LIN {X 0,Y 387.005,Z 815.122,A -85,B 0,C 180,E1 -12042.119,E2 -12042.119} C_VEL
LIN {X 0,Y 389.594,Z 822.975,A -85,B 0,C 180,E1 -12042.96,E2 -12042.96} C_VEL
LIN {X 0,Y 390.009,Z 825.761,A -85,B 0,C 180,E1 -12043.242,E2 -12043.242} C_VEL
LIN {X 0,Y 389.304,Z 834.795,A -85,B 0,C 180,E1 -12044.101,E2 -12044.101} C_VEL
LIN {X 0,Y 388.401,Z 845.399,A -85,B 0,C 180,E1 -12045.326,E2 -12045.326} C_VEL
LIN {X 0,Y 387.347,Z 856.042,A -85,B 0,C 180,E1 -12046.891,E2 -12046.891} C_VEL
LIN {X 0,Y 386.493,Z 863.14,A -85,B 0,C 180,E1 -12048.196,E2 -12048.196} C_VEL
LIN {X 0,Y 385.858,Z 869.08,A -85,B 0,C 180,E1 -12049.506,E2 -12049.506} C_VEL
LIN {X 0,Y 385.357,Z 873.167,A -85,B 0,C 180,E1 -12050.553,E2 -12050.553} C_VEL
LIN {X 0,Y 384.731,Z 878.114,A -85,B 0,C 180,E1 -12052.125,E2 -12052.125} C_VEL
LIN {X 0,Y 383.96,Z 881.899,A -85,B 0,C 180,E1 -12053.695,E2 -12053.695} C_VEL
LIN {X 0,Y 383.86,Z 883.852,A -85,B 0,C 180,E1 -12054.748,E2 -12054.748} C_VEL
LIN {X 0,Y 383.471,Z 886.332,A -85,B 0,C 180,E1 -12056.848,E2 -12056.848} C_VEL
LIN {X 0,Y 383.299,Z 887.036,A -85,B 0,C 180,E1 -12057.898,E2 -12057.898} C_VEL
LIN {X 0,Y 383.093,Z 887.297,A -85,B 0,C 180,E1 -12058.949,E2 -12058.949} C_VEL
LIN {X 0,Y 383.035,Z 886.513,A -85,B 0,C 180,E1 -12061.051,E2 -12061.051} C_VEL
LIN {X 0,Y 382.901,Z 884.089,A -85,B 0,C 180,E1 -12063.157,E2 -12063.157} C_VEL
LIN {X 0,Y 383.149,Z 881.129,A -85,B 0,C 180,E1 -12064.735,E2 -12064.735} C_VEL
LIN {X 0,Y 383.443,Z 877.126,A -85,B 0,C 180,E1 -12066.314,E2 -12066.314} C_VEL
LIN {X 0,Y 383.766,Z 871.975,A -85,B 0,C 180,E1 -12067.895,E2 -12067.895} C_VEL
LIN {X 0,Y 384.086,Z 866.854,A -85,B 0,C 180,E1 -12069.187,E2 -12069.187} C_VEL
LIN {X 0,Y 384.606,Z 859.101,A -85,B 0,C 180,E1 -12070.795,E2 -12070.795} C_VEL
LIN {X 0,Y 385.028,Z 851.181,A -85,B 0,C 180,E1 -12072.117,E2 -12072.117} C_VEL
LIN {X 0,Y 385.562,Z 843.782,A -85,B 0,C 180,E1 -12073.171,E2 -12073.171} C_VEL
LIN {X 0,Y 386.012,Z 836.271,A -85,B 0,C 180,E1 -12074.094,E2 -12074.094} C_VEL
LIN {X 0,Y 386.607,Z 826.481,A -85,B 0,C 180,E1 -12075.117,E2 -12075.117} C_VEL
LIN {X 0,Y 386.907,Z 820.016,A -85,B 0,C 180,E1 -12075.69,E2 -12075.69} C_VEL
LIN {X 0,Y 384.066,Z 808.559,A -85,B 0,C 180,E1 -12076.657,E2 -12076.657} C_VEL
LIN {X 0,Y 383.065,Z 804.769,A -85,B 0,C 180,E1 -12076.968,E2 -12076.968} C_VEL
LIN {X 0,Y 383.009,Z 804.767,A -85,B 0,C 180,E1 -12080.636,E2 -12080.636} C_VEL
LIN {X 0,Y 383.012,Z 804.777,A -85,B 0,C 180,E1 -12083.809,E2 -12083.809} C_VEL
LIN {X 0,Y 382.972,Z 804.773,A -85,B 0,C 180,E1 -12087.309,E2 -12087.309} C_VEL
LIN {X 0,Y 382.987,Z 804.773,A -85,B 0,C 180,E1 -12090.918,E2 -12090.918} C_VEL
LIN {X 0,Y 383.018,Z 804.77,A -85,B 0,C 180,E1 -12094.668,E2 -12094.668} C_VEL
LIN {X 0,Y 382.998,Z 804.772,A -85,B 0,C 180,E1 -12097.901,E2 -12097.901} C_VEL
LIN {X 0,Y 382.967,Z 804.777,A -85,B 0,C 180,E1 -12101.35,E2 -12101.35} C_VEL
LIN {X 0,Y 383,Z 804.777,A -85,B 0,C 180,E1 -12104.302,E2 -12104.302} C_VEL
LIN {X 0,Y 383.017,Z 804.77,A -85,B 0,C 180,E1 -12107.239,E2 -12107.239} C_VEL
LIN {X 0,Y 382.992,Z 804.778,A -85,B 0,C 180,E1 -12110.418,E2 -12110.418} C_VEL
LIN {X 0,Y 383.03,Z 804.773,A -85,B 0,C 180,E1 -12114.043,E2 -12114.043} C_VEL
LIN {X 0,Y 382.994,Z 804.774,A -85,B 0,C 180,E1 -12117.577,E2 -12117.577} C_VEL
LIN {X 0,Y 382.999,Z 804.774,A -85,B 0,C 180,E1 -12120.299,E2 -12120.299} C_VEL
LIN {X 0,Y 383.086,Z 804.762,A -85,B 0,C 180,E1 -12124.02,E2 -12124.02} C_VEL
LIN {X 0,Y 383.018,Z 804.772,A -85,B 0,C 180,E1 -12127.334,E2 -12127.334} C_VEL
LIN {X 0,Y 383.066,Z 804.775,A -85,B 0,C 180,E1 -12130.715,E2 -12130.715} C_VEL
LIN {X 0,Y 383.075,Z 804.773,A -85,B 0,C 180,E1 -12131.917,E2 -12131.917} C_VEL
LIN {X 0,Y 386.733,Z 816.026,A -85,B 0,C 180,E1 -12132.822,E2 -12132.822} C_VEL
LIN {X 0,Y 388.874,Z 823.669,A -85,B 0,C 180,E1 -12133.533,E2 -12133.533} C_VEL
LIN {X 0,Y 388.161,Z 834.358,A -85,B 0,C 180,E1 -12134.509,E2 -12134.509} C_VEL
LIN {X 0,Y 387.355,Z 844.687,A -85,B 0,C 180,E1 -12135.686,E2 -12135.686} C_VEL
LIN {X 0,Y 386.66,Z 853.102,A -85,B 0,C 180,E1 -12136.866,E2 -12136.866} C_VEL
LIN {X 0,Y 385.851,Z 860.859,A -85,B 0,C 180,E1 -12138.174,E2 -12138.174} C_VEL
LIN {X 0,Y 385.124,Z 868.416,A -85,B 0,C 180,E1 -12139.75,E2 -12139.75} C_VEL
LIN {X 0,Y 384.606,Z 874.215,A -85,B 0,C 180,E1 -12141.259,E2 -12141.259} C_VEL
LIN {X 0,Y 384.195,Z 878.536,A -85,B 0,C 180,E1 -12142.641,E2 -12142.641} C_VEL
LIN {X 0,Y 383.606,Z 882.429,A -85,B 0,C 180,E1 -12144.215,E2 -12144.215} C_VEL
LIN {X 0,Y 383.294,Z 885.283,A -85,B 0,C 180,E1 -12145.792,E2 -12145.792} C_VEL
LIN {X 0,Y 383.255,Z 886.638,A -85,B 0,C 180,E1 -12146.845,E2 -12146.845} C_VEL
LIN {X 0,Y 383.14,Z 888.204,A -85,B 0,C 180,E1 -12148.947,E2 -12148.947} C_VEL
LIN {X 0,Y 383.115,Z 888.434,A -85,B 0,C 180,E1 -12149.998,E2 -12149.998} C_VEL
LIN {X 0,Y 383.209,Z 887.68,A -85,B 0,C 180,E1 -12152.1,E2 -12152.1} C_VEL
LIN {X 0,Y 383.284,Z 885.44,A -85,B 0,C 180,E1 -12154.204,E2 -12154.204} C_VEL
LIN {X 0,Y 383.597,Z 882.636,A -85,B 0,C 180,E1 -12155.781,E2 -12155.781} C_VEL
LIN {X 0,Y 384.207,Z 878.803,A -85,B 0,C 180,E1 -12157.355,E2 -12157.355} C_VEL
LIN {X 0,Y 384.759,Z 873.232,A -85,B 0,C 180,E1 -12159.118,E2 -12159.118} C_VEL
LIN {X 0,Y 385.332,Z 866.527,A -85,B 0,C 180,E1 -12160.773,E2 -12160.773} C_VEL
LIN {X 0,Y 386.172,Z 858.507,A -85,B 0,C 180,E1 -12162.345,E2 -12162.345} C_VEL
LIN {X 0,Y 386.907,Z 850.291,A -85,B 0,C 180,E1 -12163.657,E2 -12163.657} C_VEL
LIN {X 0,Y 387.698,Z 840.121,A -85,B 0,C 180,E1 -12164.968,E2 -12164.968} C_VEL
LIN {X 0,Y 388.537,Z 830.16,A -85,B 0,C 180,E1 -12165.996,E2 -12165.996} C_VEL
LIN {X 0,Y 388.94,Z 824.397,A -85,B 0,C 180,E1 -12166.5,E2 -12166.5} C_VEL
LIN {X 0,Y 386.451,Z 815.179,A -85,B 0,C 180,E1 -12167.353,E2 -12167.353} C_VEL
LIN {X 0,Y 383.347,Z 805.87,A -85,B 0,C 180,E1 -12168.103,E2 -12168.103} C_VEL
LIN {X 0,Y 382.713,Z 804.974,A -85,B 0,C 180,E1 -12168.303,E2 -12168.303} C_VEL
LIN {X 0,Y 378.642,Z 805.321,A -85,B 0,C 180,E1 -12170.049,E2 -12170.049} C_VEL
LIN {X 0,Y 377.112,Z 805.902,A -85,B 0,C 180,E1 -12171.038,E2 -12171.038} C_VEL
LIN {X 0,Y 376.15,Z 805.753,A -85,B 0,C 180,E1 -12172.053,E2 -12172.053} C_VEL
LIN {X 0,Y 375.966,Z 805.649,A -85,B 0,C 180,E1 -12172.738,E2 -12172.738} C_VEL
LIN {X 0,Y 376.037,Z 805.646,A -85,B 0,C 180,E1 -12176.22,E2 -12176.22} C_VEL
LIN {X 0,Y 375.965,Z 805.652,A -85,B 0,C 180,E1 -12179.077,E2 -12179.077} C_VEL
LIN {X 0,Y 375.945,Z 805.654,A -85,B 0,C 180,E1 -12182.826,E2 -12182.826} C_VEL
LIN {X 0,Y 375.951,Z 805.654,A -85,B 0,C 180,E1 -12185.413,E2 -12185.413} C_VEL
LIN {X 0,Y 375.97,Z 805.656,A -85,B 0,C 180,E1 -12188.269,E2 -12188.269} C_VEL
LIN {X 0,Y 375.98,Z 805.649,A -85,B 0,C 180,E1 -12191.608,E2 -12191.608} C_VEL
LIN {X 0,Y 376.006,Z 805.645,A -85,B 0,C 180,E1 -12195.253,E2 -12195.253} C_VEL
LIN {X 0,Y 375.989,Z 805.648,A -85,B 0,C 180,E1 -12199.139,E2 -12199.139} C_VEL
LIN {X 0,Y 375.961,Z 805.647,A -85,B 0,C 180,E1 -12201.911,E2 -12201.911} C_VEL
LIN {X 0,Y 375.967,Z 805.645,A -85,B 0,C 180,E1 -12205.331,E2 -12205.331} C_VEL
LIN {X 0,Y 375.946,Z 805.656,A -85,B 0,C 180,E1 -12208.437,E2 -12208.437} C_VEL
LIN {X 0,Y 375.988,Z 805.648,A -85,B 0,C 180,E1 -12212.14,E2 -12212.14} C_VEL
LIN {X 0,Y 375.991,Z 805.647,A -85,B 0,C 180,E1 -12214.538,E2 -12214.538} C_VEL
LIN {X 0,Y 375.947,Z 805.651,A -85,B 0,C 180,E1 -12218.045,E2 -12218.045} C_VEL
LIN {X 0,Y 375.993,Z 805.649,A -85,B 0,C 180,E1 -12221.472,E2 -12221.472} C_VEL
LIN {X 0,Y 376.043,Z 805.637,A -85,B 0,C 180,E1 -12224.832,E2 -12224.832} C_VEL
LIN {X 0,Y 376.044,Z 805.641,A -85,B 0,C 180,E1 -12228.136,E2 -12228.136} C_VEL
LIN {X 0,Y 376.202,Z 805.622,A -85,B 0,C 180,E1 -12231.918,E2 -12231.918} C_VEL
LIN {X 0,Y 376.152,Z 805.63,A -85,B 0,C 180,E1 -12234.64,E2 -12234.64} C_VEL
LIN {X 0,Y 376.336,Z 805.608,A -85,B 0,C 180,E1 -12237.859,E2 -12237.859} C_VEL
LIN {X 0,Y 376.471,Z 805.592,A -85,B 0,C 180,E1 -12240,E2 -12240} C_VEL
LIN {X 0,Y 376.168,Z 805.631,A -85,B 0,C 180,E1 -12243.213,E2 -12243.213} C_VEL
LIN {X 0,Y 376.202,Z 805.62,A -85,B 0,C 180,E1 -12246.436,E2 -12246.436} C_VEL
LIN {X 0,Y 376.106,Z 805.638,A -85,B 0,C 180,E1 -12249.682,E2 -12249.682} C_VEL
LIN {X 0,Y 376.073,Z 805.637,A -85,B 0,C 180,E1 -12253.659,E2 -12253.659} C_VEL
LIN {X 0,Y 376.027,Z 805.647,A -85,B 0,C 180,E1 -12257.608,E2 -12257.608} C_VEL
LIN {X 0,Y 375.962,Z 805.652,A -85,B 0,C 180,E1 -12260.833,E2 -12260.833} C_VEL
LIN {X 0,Y 375.946,Z 805.657,A -85,B 0,C 180,E1 -12264.285,E2 -12264.285} C_VEL
LIN {X 0,Y 375.919,Z 805.656,A -85,B 0,C 180,E1 -12267.865,E2 -12267.865} C_VEL
LIN {X 0,Y 375.942,Z 805.655,A -85,B 0,C 180,E1 -12271.564,E2 -12271.564} C_VEL
LIN {X 0,Y 375.934,Z 805.656,A -85,B 0,C 180,E1 -12275.418,E2 -12275.418} C_VEL
LIN {X 0,Y 375.921,Z 805.66,A -85,B 0,C 180,E1 -12278.264,E2 -12278.264} C_VEL
LIN {X 0,Y 375.902,Z 805.658,A -85,B 0,C 180,E1 -12281.599,E2 -12281.599} C_VEL
LIN {X 0,Y 375.973,Z 805.715,A -85,B 0,C 180,E1 -12284.647,E2 -12284.647} C_VEL
LIN {X 0,Y 377.826,Z 814.71,A -85,B 0,C 180,E1 -12288.077,E2 -12288.077} C_VEL
LIN {X 0,Y 379.425,Z 823.13,A -85,B 0,C 180,E1 -12291.074,E2 -12291.074} C_VEL
LIN {X 0,Y 380.127,Z 827.814,A -85,B 0,C 180,E1 -12292.656,E2 -12292.656} C_VEL
LIN {X 0,Y 379.363,Z 836.21,A -85,B 0,C 180,E1 -12295.276,E2 -12295.276} C_VEL
LIN {X 0,Y 378.494,Z 846.362,A -85,B 0,C 180,E1 -12298.364,E2 -12298.364} C_VEL
LIN {X 0,Y 377.529,Z 858.416,A -85,B 0,C 180,E1 -12301.965,E2 -12301.965} C_VEL
LIN {X 0,Y 376.671,Z 871.275,A -85,B 0,C 180,E1 -12305.768,E2 -12305.768} C_VEL
LIN {X 0,Y 375.923,Z 884.784,A -85,B 0,C 180,E1 -12309.768,E2 -12309.768} C_VEL
LIN {X 0,Y 375.758,Z 887.708,A -85,B 0,C 180,E1 -12310.649,E2 -12310.649} C_VEL
LIN {X 0,Y 377.592,Z 902.844,A -85,B 0,C 180,E1 -12311.226,E2 -12311.226} C_VEL
LIN {X 0,Y 378.505,Z 914.998,A -85,B 0,C 180,E1 -12311.859,E2 -12311.859} C_VEL
LIN {X 0,Y 378.99,Z 926.426,A -85,B 0,C 180,E1 -12312.629,E2 -12312.629} C_VEL
LIN {X 0,Y 379.31,Z 933.112,A -85,B 0,C 180,E1 -12313.174,E2 -12313.174} C_VEL
LIN {X 0,Y 378.282,Z 944.543,A -85,B 0,C 180,E1 -12314.236,E2 -12314.236} C_VEL
LIN {X 0,Y 377.374,Z 954.899,A -85,B 0,C 180,E1 -12315.441,E2 -12315.441} C_VEL
LIN {X 0,Y 376.873,Z 960.709,A -85,B 0,C 180,E1 -12316.248,E2 -12316.248} C_VEL
LIN {X 0,Y 376.057,Z 970.58,A -85,B 0,C 180,E1 -12317.865,E2 -12317.865} C_VEL
LIN {X 0,Y 375.481,Z 978.479,A -85,B 0,C 180,E1 -12319.487,E2 -12319.487} C_VEL
LIN {X 0,Y 375.258,Z 983.922,A -85,B 0,C 180,E1 -12320.842,E2 -12320.842} C_VEL
LIN {X 0,Y 375.127,Z 989.217,A -85,B 0,C 180,E1 -12322.466,E2 -12322.466} C_VEL
LIN {X 0,Y 375.135,Z 993.353,A -85,B 0,C 180,E1 -12324.088,E2 -12324.088} C_VEL
LIN {X 0,Y 375.31,Z 996.435,A -85,B 0,C 180,E1 -12325.706,E2 -12325.706} C_VEL
LIN {X 0,Y 375.302,Z 997.888,A -85,B 0,C 180,E1 -12326.781,E2 -12326.781} C_VEL
LIN {X 0,Y 375.322,Z 998.927,A -85,B 0,C 180,E1 -12327.856,E2 -12327.856} C_VEL
LIN {X 0,Y 375.36,Z 999.564,A -85,B 0,C 180,E1 -12328.929,E2 -12328.929} C_VEL
LIN {X 0,Y 375.391,Z 999.792,A -85,B 0,C 180,E1 -12330.002,E2 -12330.002} C_VEL
LIN {X 0,Y 375.361,Z 999.56,A -85,B 0,C 180,E1 -12331.075,E2 -12331.075} C_VEL
LIN {X 0,Y 375.323,Z 998.92,A -85,B 0,C 180,E1 -12332.148,E2 -12332.148} C_VEL
LIN {X 0,Y 375.303,Z 997.876,A -85,B 0,C 180,E1 -12333.222,E2 -12333.222} C_VEL
LIN {X 0,Y 375.311,Z 996.419,A -85,B 0,C 180,E1 -12334.298,E2 -12334.298} C_VEL
LIN {X 0,Y 375.132,Z 993.334,A -85,B 0,C 180,E1 -12335.916,E2 -12335.916} C_VEL
LIN {X 0,Y 375.129,Z 989.196,A -85,B 0,C 180,E1 -12337.538,E2 -12337.538} C_VEL
LIN {X 0,Y 375.292,Z 982.856,A -85,B 0,C 180,E1 -12339.433,E2 -12339.433} C_VEL
LIN {X 0,Y 375.639,Z 975.971,A -85,B 0,C 180,E1 -12341.058,E2 -12341.058} C_VEL
LIN {X 0,Y 376.257,Z 967.476,A -85,B 0,C 180,E1 -12342.68,E2 -12342.68} C_VEL
LIN {X 0,Y 376.939,Z 960.656,A -85,B 0,C 180,E1 -12343.754,E2 -12343.754} C_VEL
LIN {X 0,Y 377.733,Z 950.483,A -85,B 0,C 180,E1 -12345.1,E2 -12345.1} C_VEL
LIN {X 0,Y 378.682,Z 940.495,A -85,B 0,C 180,E1 -12346.166,E2 -12346.166} C_VEL
LIN {X 0,Y 379.363,Z 931.379,A -85,B 0,C 180,E1 -12346.966,E2 -12346.966} C_VEL
LIN {X 0,Y 378.707,Z 919.645,A -85,B 0,C 180,E1 -12347.845,E2 -12347.845} C_VEL
LIN {X 0,Y 376.989,Z 894.092,A -85,B 0,C 180,E1 -12349.316,E2 -12349.316} C_VEL
LIN {X 0,Y 375.865,Z 886.401,A -85,B 0,C 180,E1 -12349.741,E2 -12349.741} C_VEL
LIN {X 0,Y 376.59,Z 872.485,A -85,B 0,C 180,E1 -12353.872,E2 -12353.872} C_VEL
LIN {X 0,Y 377.465,Z 859.373,A -85,B 0,C 180,E1 -12357.743,E2 -12357.743} C_VEL
LIN {X 0,Y 378.602,Z 845.303,A -85,B 0,C 180,E1 -12361.943,E2 -12361.943} C_VEL
LIN {X 0,Y 379.636,Z 833.778,A -85,B 0,C 180,E1 -12365.457,E2 -12365.457} C_VEL
LIN {X 0,Y 380.069,Z 827.797,A -85,B 0,C 180,E1 -12367.332,E2 -12367.332} C_VEL
LIN {X 0,Y 378.949,Z 820.743,A -85,B 0,C 180,E1 -12369.739,E2 -12369.739} C_VEL
LIN {X 0,Y 377.34,Z 812.535,A -85,B 0,C 180,E1 -12372.713,E2 -12372.713} C_VEL
LIN {X 0,Y 375.913,Z 805.662,A -85,B 0,C 180,E1 -12375.432,E2 -12375.432} C_VEL
LIN {X 0,Y 375.914,Z 805.661,A -85,B 0,C 180,E1 -12379.129,E2 -12379.129} C_VEL
LIN {X 0,Y 375.954,Z 805.655,A -85,B 0,C 180,E1 -12381.91,E2 -12381.91} C_VEL
LIN {X 0,Y 375.977,Z 805.651,A -85,B 0,C 180,E1 -12385.335,E2 -12385.335} C_VEL
LIN {X 0,Y 375.958,Z 805.656,A -85,B 0,C 180,E1 -12388.438,E2 -12388.438} C_VEL
LIN {X 0,Y 375.921,Z 805.659,A -85,B 0,C 180,E1 -12392.135,E2 -12392.135} C_VEL
LIN {X 0,Y 375.934,Z 805.659,A -85,B 0,C 180,E1 -12394.534,E2 -12394.534} C_VEL
LIN {X 0,Y 375.972,Z 805.652,A -85,B 0,C 180,E1 -12396.887,E2 -12396.887} C_VEL
LIN {X 0,Y 375.961,Z 805.656,A -85,B 0,C 180,E1 -12400.495,E2 -12400.495} C_VEL
LIN {X 0,Y 377.057,Z 808.624,A -85,B 0,C 180,E1 -12400.799,E2 -12400.799} C_VEL
LIN {X 0,Y 380.901,Z 818.112,A -85,B 0,C 180,E1 -12401.822,E2 -12401.822} C_VEL
LIN {X 0,Y 383.447,Z 826.235,A -85,B 0,C 180,E1 -12402.744,E2 -12402.744} C_VEL
LIN {X 0,Y 383.122,Z 833.12,A -85,B 0,C 180,E1 -12403.403,E2 -12403.403} C_VEL
LIN {X 0,Y 382.335,Z 842.18,A -85,B 0,C 180,E1 -12404.405,E2 -12404.405} C_VEL
LIN {X 0,Y 381.597,Z 849.325,A -85,B 0,C 180,E1 -12405.331,E2 -12405.331} C_VEL
LIN {X 0,Y 380.665,Z 857.926,A -85,B 0,C 180,E1 -12406.657,E2 -12406.657} C_VEL
LIN {X 0,Y 379.759,Z 864.878,A -85,B 0,C 180,E1 -12407.983,E2 -12407.983} C_VEL
LIN {X 0,Y 379.063,Z 870.716,A -85,B 0,C 180,E1 -12409.315,E2 -12409.315} C_VEL
LIN {X 0,Y 378.525,Z 874.719,A -85,B 0,C 180,E1 -12410.381,E2 -12410.381} C_VEL
LIN {X 0,Y 377.872,Z 879.591,A -85,B 0,C 180,E1 -12411.982,E2 -12411.982} C_VEL
LIN {X 0,Y 377.065,Z 883.279,A -85,B 0,C 180,E1 -12413.579,E2 -12413.579} C_VEL
LIN {X 0,Y 376.918,Z 885.208,A -85,B 0,C 180,E1 -12414.651,E2 -12414.651} C_VEL
LIN {X 0,Y 376.507,Z 887.57,A -85,B 0,C 180,E1 -12416.79,E2 -12416.79} C_VEL
LIN {X 0,Y 376.32,Z 888.249,A -85,B 0,C 180,E1 -12417.859,E2 -12417.859} C_VEL
LIN {X 0,Y 376.089,Z 888.445,A -85,B 0,C 180,E1 -12418.929,E2 -12418.929} C_VEL
LIN {X 0,Y 376.021,Z 887.579,A -85,B 0,C 180,E1 -12421.071,E2 -12421.071} C_VEL
LIN {X 0,Y 375.875,Z 885.032,A -85,B 0,C 180,E1 -12423.216,E2 -12423.216} C_VEL
LIN {X 0,Y 376.142,Z 881.988,A -85,B 0,C 180,E1 -12424.823,E2 -12424.823} C_VEL
LIN {X 0,Y 376.453,Z 879.437,A -85,B 0,C 180,E1 -12425.894,E2 -12425.894} C_VEL
LIN {X 0,Y 376.661,Z 874.632,A -85,B 0,C 180,E1 -12427.505,E2 -12427.505} C_VEL
LIN {X 0,Y 377.108,Z 867.44,A -85,B 0,C 180,E1 -12429.358,E2 -12429.358} C_VEL
LIN {X 0,Y 377.659,Z 859.595,A -85,B 0,C 180,E1 -12430.996,E2 -12430.996} C_VEL
LIN {X 0,Y 378.223,Z 849.823,A -85,B 0,C 180,E1 -12432.611,E2 -12432.611} C_VEL
LIN {X 0,Y 379,Z 838.755,A -85,B 0,C 180,E1 -12434.086,E2 -12434.086} C_VEL
LIN {X 0,Y 379.715,Z 826.985,A -85,B 0,C 180,E1 -12435.343,E2 -12435.343} C_VEL
LIN {X 0,Y 379.953,Z 821.075,A -85,B 0,C 180,E1 -12435.875,E2 -12435.875} C_VEL
LIN {X 0,Y 376.925,Z 809.093,A -85,B 0,C 180,E1 -12436.903,E2 -12436.903} C_VEL
LIN {X 0,Y 376.009,Z 805.649,A -85,B 0,C 180,E1 -12437.191,E2 -12437.191} C_VEL
LIN {X 0,Y 375.952,Z 805.646,A -85,B 0,C 180,E1 -12440.818,E2 -12440.818} C_VEL
LIN {X 0,Y 375.94,Z 805.653,A -85,B 0,C 180,E1 -12444.285,E2 -12444.285} C_VEL
LIN {X 0,Y 375.915,Z 805.65,A -85,B 0,C 180,E1 -12446.66,E2 -12446.66} C_VEL
LIN {X 0,Y 375.919,Z 805.653,A -85,B 0,C 180,E1 -12449.084,E2 -12449.084} C_VEL
LIN {X 0,Y 375.963,Z 805.652,A -85,B 0,C 180,E1 -12451.562,E2 -12451.562} C_VEL
LIN {X 0,Y 375.955,Z 805.651,A -85,B 0,C 180,E1 -12455.416,E2 -12455.416} C_VEL
LIN {X 0,Y 375.94,Z 805.653,A -85,B 0,C 180,E1 -12458.262,E2 -12458.262} C_VEL
LIN {X 0,Y 375.923,Z 805.656,A -85,B 0,C 180,E1 -12461.597,E2 -12461.597} C_VEL
LIN {X 0,Y 375.932,Z 805.654,A -85,B 0,C 180,E1 -12464.73,E2 -12464.73} C_VEL
LIN {X 0,Y 375.932,Z 805.656,A -85,B 0,C 180,E1 -12467.698,E2 -12467.698} C_VEL
LIN {X 0,Y 375.941,Z 805.656,A -85,B 0,C 180,E1 -12470.533,E2 -12470.533} C_VEL
LIN {X 0,Y 375.969,Z 805.647,A -85,B 0,C 180,E1 -12473.495,E2 -12473.495} C_VEL
LIN {X 0,Y 375.967,Z 805.653,A -85,B 0,C 180,E1 -12475.888,E2 -12475.888} C_VEL
LIN {X 0,Y 375.971,Z 805.647,A -85,B 0,C 180,E1 -12479.686,E2 -12479.686} C_VEL
LIN {X 0,Y 376.026,Z 805.638,A -85,B 0,C 180,E1 -12483.347,E2 -12483.347} C_VEL
LIN {X 0,Y 376.004,Z 805.648,A -85,B 0,C 180,E1 -12486.887,E2 -12486.887} C_VEL
LIN {X 0,Y 376.004,Z 805.654,A -85,B 0,C 180,E1 -12490.338,E2 -12490.338} C_VEL
LIN {X 0,Y 376.025,Z 805.65,A -85,B 0,C 180,E1 -12491.55,E2 -12491.55} C_VEL
LIN {X 0,Y 380.249,Z 818.59,A -85,B 0,C 180,E1 -12492.631,E2 -12492.631} C_VEL
LIN {X 0,Y 382.168,Z 826.388,A -85,B 0,C 180,E1 -12493.386,E2 -12493.386} C_VEL
LIN {X 0,Y 381.292,Z 836.665,A -85,B 0,C 180,E1 -12494.36,E2 -12494.36} C_VEL
LIN {X 0,Y 380.478,Z 846.766,A -85,B 0,C 180,E1 -12495.558,E2 -12495.558} C_VEL
LIN {X 0,Y 379.674,Z 855.808,A -85,B 0,C 180,E1 -12496.892,E2 -12496.892} C_VEL
LIN {X 0,Y 378.732,Z 864.579,A -85,B 0,C 180,E1 -12498.491,E2 -12498.491} C_VEL
LIN {X 0,Y 378.015,Z 871.977,A -85,B 0,C 180,E1 -12500.189,E2 -12500.189} C_VEL
LIN {X 0,Y 377.424,Z 878.008,A -85,B 0,C 180,E1 -12501.97,E2 -12501.97} C_VEL
LIN {X 0,Y 376.712,Z 882.271,A -85,B 0,C 180,E1 -12503.571,E2 -12503.571} C_VEL
LIN {X 0,Y 376.502,Z 884.496,A -85,B 0,C 180,E1 -12504.643,E2 -12504.643} C_VEL
LIN {X 0,Y 376.289,Z 886.315,A -85,B 0,C 180,E1 -12505.714,E2 -12505.714} C_VEL
LIN {X 0,Y 376.241,Z 887.67,A -85,B 0,C 180,E1 -12506.786,E2 -12506.786} C_VEL
LIN {X 0,Y 376.121,Z 889.235,A -85,B 0,C 180,E1 -12508.927,E2 -12508.927} C_VEL
LIN {X 0,Y 376.092,Z 889.465,A -85,B 0,C 180,E1 -12509.998,E2 -12509.998} C_VEL
LIN {X 0,Y 376.198,Z 888.709,A -85,B 0,C 180,E1 -12512.139,E2 -12512.139} C_VEL
LIN {X 0,Y 376.279,Z 886.471,A -85,B 0,C 180,E1 -12514.283,E2 -12514.283} C_VEL
LIN {X 0,Y 376.608,Z 883.667,A -85,B 0,C 180,E1 -12515.889,E2 -12515.889} C_VEL
LIN {X 0,Y 377.245,Z 879.832,A -85,B 0,C 180,E1 -12517.491,E2 -12517.491} C_VEL
LIN {X 0,Y 377.827,Z 874.242,A -85,B 0,C 180,E1 -12519.292,E2 -12519.292} C_VEL
LIN {X 0,Y 378.433,Z 867.556,A -85,B 0,C 180,E1 -12520.971,E2 -12520.971} C_VEL
LIN {X 0,Y 379.313,Z 859.536,A -85,B 0,C 180,E1 -12522.572,E2 -12522.572} C_VEL
LIN {X 0,Y 380.084,Z 851.319,A -85,B 0,C 180,E1 -12523.907,E2 -12523.907} C_VEL
LIN {X 0,Y 380.916,Z 841.148,A -85,B 0,C 180,E1 -12525.241,E2 -12525.241} C_VEL
LIN {X 0,Y 381.884,Z 830.362,A -85,B 0,C 180,E1 -12526.363,E2 -12526.363} C_VEL
LIN {X 0,Y 382.167,Z 825.674,A -85,B 0,C 180,E1 -12526.779,E2 -12526.779} C_VEL
LIN {X 0,Y 379.139,Z 815.139,A -85,B 0,C 180,E1 -12527.782,E2 -12527.782} C_VEL
LIN {X 0,Y 376.03,Z 805.645,A -85,B 0,C 180,E1 -12528.559,E2 -12528.559} C_VEL
LIN {X 0,Y 375.96,Z 805.654,A -85,B 0,C 180,E1 -12531.952,E2 -12531.952} C_VEL
LIN {X 0,Y 375.966,Z 805.649,A -85,B 0,C 180,E1 -12532.738,E2 -12532.738} C_VEL
LIN {X 0,Y 375.342,Z 805.733,A -85,B 0,C 180,E1 -12533.632,E2 -12533.632} C_VEL
LIN {X 0,Y 372.516,Z 806.083,A -85,B 0,C 180,E1 -12535.087,E2 -12535.087} C_VEL
LIN {X 0,Y 370.092,Z 806.386,A -85,B 0,C 180,E1 -12536.263,E2 -12536.263} C_VEL
LIN {X 0,Y 369.041,Z 806.514,A -85,B 0,C 180,E1 -12537.173,E2 -12537.173} C_VEL
LIN {X 0,Y 368.951,Z 806.524,A -85,B 0,C 180,E1 -12537.481,E2 -12537.481} C_VEL
LIN {X 0,Y 368.904,Z 806.531,A -85,B 0,C 180,E1 -12540.985,E2 -12540.985} C_VEL
LIN {X 0,Y 368.93,Z 806.528,A -85,B 0,C 180,E1 -12544.851,E2 -12544.851} C_VEL
LIN {X 0,Y 368.905,Z 806.533,A -85,B 0,C 180,E1 -12548.639,E2 -12548.639} C_VEL
LIN {X 0,Y 368.942,Z 806.529,A -85,B 0,C 180,E1 -12552.019,E2 -12552.019} C_VEL
LIN {X 0,Y 368.98,Z 806.521,A -85,B 0,C 180,E1 -12555.191,E2 -12555.191} C_VEL
LIN {X 0,Y 368.93,Z 806.526,A -85,B 0,C 180,E1 -12558.184,E2 -12558.184} C_VEL
LIN {X 0,Y 368.904,Z 806.525,A -85,B 0,C 180,E1 -12561.356,E2 -12561.356} C_VEL
LIN {X 0,Y 368.924,Z 806.523,A -85,B 0,C 180,E1 -12565.145,E2 -12565.145} C_VEL
LIN {X 0,Y 368.915,Z 806.527,A -85,B 0,C 180,E1 -12569.045,E2 -12569.045} C_VEL
LIN {X 0,Y 368.972,Z 806.521,A -85,B 0,C 180,E1 -12571.563,E2 -12571.563} C_VEL
LIN {X 0,Y 368.943,Z 806.527,A -85,B 0,C 180,E1 -12575.223,E2 -12575.223} C_VEL
LIN {X 0,Y 368.922,Z 806.528,A -85,B 0,C 180,E1 -12578.972,E2 -12578.972} C_VEL
LIN {X 0,Y 368.974,Z 806.521,A -85,B 0,C 180,E1 -12582.256,E2 -12582.256} C_VEL
LIN {X 0,Y 369.021,Z 806.513,A -85,B 0,C 180,E1 -12586.227,E2 -12586.227} C_VEL
LIN {X 0,Y 369.056,Z 806.507,A -85,B 0,C 180,E1 -12590.131,E2 -12590.131} C_VEL
LIN {X 0,Y 369.145,Z 806.5,A -85,B 0,C 180,E1 -12592.341,E2 -12592.341} C_VEL
LIN {X 0,Y 369.125,Z 806.506,A -85,B 0,C 180,E1 -12594.537,E2 -12594.537} C_VEL
LIN {X 0,Y 369.301,Z 806.485,A -85,B 0,C 180,E1 -12597.819,E2 -12597.819} C_VEL
LIN {X 0,Y 369.44,Z 806.468,A -85,B 0,C 180,E1 -12600,E2 -12600} C_VEL
LIN {X 0,Y 369.299,Z 806.484,A -85,B 0,C 180,E1 -12602.181,E2 -12602.181} C_VEL
LIN {X 0,Y 369.164,Z 806.497,A -85,B 0,C 180,E1 -12606.559,E2 -12606.559} C_VEL
LIN {X 0,Y 369.105,Z 806.504,A -85,B 0,C 180,E1 -12608.762,E2 -12608.762} C_VEL
LIN {X 0,Y 368.995,Z 806.516,A -85,B 0,C 180,E1 -12612.094,E2 -12612.094} C_VEL
LIN {X 0,Y 368.981,Z 806.524,A -85,B 0,C 180,E1 -12615.466,E2 -12615.466} C_VEL
LIN {X 0,Y 368.95,Z 806.526,A -85,B 0,C 180,E1 -12618.895,E2 -12618.895} C_VEL
LIN {X 0,Y 368.905,Z 806.534,A -85,B 0,C 180,E1 -12622.397,E2 -12622.397} C_VEL
LIN {X 0,Y 368.909,Z 806.534,A -85,B 0,C 180,E1 -12625.987,E2 -12625.987} C_VEL
LIN {X 0,Y 368.881,Z 806.536,A -85,B 0,C 180,E1 -12629.693,E2 -12629.693} C_VEL
LIN {X 0,Y 368.882,Z 806.534,A -85,B 0,C 180,E1 -12633.044,E2 -12633.044} C_VEL
LIN {X 0,Y 368.897,Z 806.536,A -85,B 0,C 180,E1 -12636.199,E2 -12636.199} C_VEL
LIN {X 0,Y 368.86,Z 806.54,A -85,B 0,C 180,E1 -12638.959,E2 -12638.959} C_VEL
LIN {X 0,Y 368.851,Z 806.534,A -85,B 0,C 180,E1 -12642.008,E2 -12642.008} C_VEL
LIN {X 0,Y 368.93,Z 806.645,A -85,B 0,C 180,E1 -12644.245,E2 -12644.245} C_VEL
LIN {X 0,Y 370.974,Z 816.509,A -85,B 0,C 180,E1 -12648.08,E2 -12648.08} C_VEL
LIN {X 0,Y 372.749,Z 826.067,A -85,B 0,C 180,E1 -12651.526,E2 -12651.526} C_VEL
LIN {X 0,Y 373.152,Z 830.232,A -85,B 0,C 180,E1 -12652.94,E2 -12652.94} C_VEL
LIN {X 0,Y 371.859,Z 843.406,A -85,B 0,C 180,E1 -12657.09,E2 -12657.09} C_VEL
LIN {X 0,Y 370.664,Z 856.755,A -85,B 0,C 180,E1 -12661.186,E2 -12661.186} C_VEL
LIN {X 0,Y 369.819,Z 868.303,A -85,B 0,C 180,E1 -12664.688,E2 -12664.688} C_VEL
LIN {X 0,Y 368.964,Z 882.411,A -85,B 0,C 180,E1 -12668.963,E2 -12668.963} C_VEL
LIN {X 0,Y 368.784,Z 886.645,A -85,B 0,C 180,E1 -12670.268,E2 -12670.268} C_VEL
LIN {X 0,Y 370.645,Z 902.274,A -85,B 0,C 180,E1 -12670.88,E2 -12670.88} C_VEL
LIN {X 0,Y 371.595,Z 915.131,A -85,B 0,C 180,E1 -12671.583,E2 -12671.583} C_VEL
LIN {X 0,Y 372.044,Z 926.843,A -85,B 0,C 180,E1 -12672.41,E2 -12672.41} C_VEL
LIN {X 0,Y 372.348,Z 933.668,A -85,B 0,C 180,E1 -12672.991,E2 -12672.991} C_VEL
LIN {X 0,Y 371.28,Z 944.778,A -85,B 0,C 180,E1 -12674.072,E2 -12674.072} C_VEL
LIN {X 0,Y 370.255,Z 955.539,A -85,B 0,C 180,E1 -12675.394,E2 -12675.394} C_VEL
LIN {X 0,Y 369.793,Z 961.611,A -85,B 0,C 180,E1 -12676.278,E2 -12676.278} C_VEL
LIN {X 0,Y 369.042,Z 969.529,A -85,B 0,C 180,E1 -12677.631,E2 -12677.631} C_VEL
LIN {X 0,Y 368.443,Z 977.429,A -85,B 0,C 180,E1 -12679.284,E2 -12679.284} C_VEL
LIN {X 0,Y 368.153,Z 984.76,A -85,B 0,C 180,E1 -12681.218,E2 -12681.218} C_VEL
LIN {X 0,Y 368.065,Z 990.447,A -85,B 0,C 180,E1 -12683.176,E2 -12683.176} C_VEL
LIN {X 0,Y 368.099,Z 993.432,A -85,B 0,C 180,E1 -12684.524,E2 -12684.524} C_VEL
LIN {X 0,Y 368.243,Z 995.395,A -85,B 0,C 180,E1 -12685.624,E2 -12685.624} C_VEL
LIN {X 0,Y 368.26,Z 996.853,A -85,B 0,C 180,E1 -12686.72,E2 -12686.72} C_VEL
LIN {X 0,Y 368.286,Z 997.894,A -85,B 0,C 180,E1 -12687.815,E2 -12687.815} C_VEL
LIN {X 0,Y 368.33,Z 998.532,A -85,B 0,C 180,E1 -12688.909,E2 -12688.909} C_VEL
LIN {X 0,Y 368.366,Z 998.76,A -85,B 0,C 180,E1 -12690.002,E2 -12690.002} C_VEL
LIN {X 0,Y 368.331,Z 998.528,A -85,B 0,C 180,E1 -12691.095,E2 -12691.095} C_VEL
LIN {X 0,Y 368.287,Z 997.886,A -85,B 0,C 180,E1 -12692.189,E2 -12692.189} C_VEL
LIN {X 0,Y 368.261,Z 996.841,A -85,B 0,C 180,E1 -12693.284,E2 -12693.284} C_VEL
LIN {X 0,Y 368.244,Z 995.378,A -85,B 0,C 180,E1 -12694.38,E2 -12694.38} C_VEL
LIN {X 0,Y 368.081,Z 992.293,A -85,B 0,C 180,E1 -12696.03,E2 -12696.03} C_VEL
LIN {X 0,Y 368.072,Z 988.15,A -85,B 0,C 180,E1 -12697.683,E2 -12697.683} C_VEL
LIN {X 0,Y 368.257,Z 981.808,A -85,B 0,C 180,E1 -12699.615,E2 -12699.615} C_VEL
LIN {X 0,Y 368.631,Z 974.921,A -85,B 0,C 180,E1 -12701.271,E2 -12701.271} C_VEL
LIN {X 0,Y 369.29,Z 966.426,A -85,B 0,C 180,E1 -12702.923,E2 -12702.923} C_VEL
LIN {X 0,Y 370.065,Z 957.748,A -85,B 0,C 180,E1 -12704.295,E2 -12704.295} C_VEL
LIN {X 0,Y 371.039,Z 947.071,A -85,B 0,C 180,E1 -12705.661,E2 -12705.661} C_VEL
LIN {X 0,Y 372.138,Z 936.563,A -85,B 0,C 180,E1 -12706.74,E2 -12706.74} C_VEL
LIN {X 0,Y 372.284,Z 930.287,A -85,B 0,C 180,E1 -12707.299,E2 -12707.299} C_VEL
LIN {X 0,Y 371.749,Z 919.172,A -85,B 0,C 180,E1 -12708.152,E2 -12708.152} C_VEL
LIN {X 0,Y 370.75,Z 898.88,A -85,B 0,C 180,E1 -12709.477,E2 -12709.477} C_VEL
LIN {X 0,Y 369.269,Z 887.958,A -85,B 0,C 180,E1 -12710.125,E2 -12710.125} C_VEL
LIN {X 0,Y 368.85,Z 884.692,A -85,B 0,C 180,E1 -12710.334,E2 -12710.334} C_VEL
LIN {X 0,Y 369.705,Z 870.242,A -85,B 0,C 180,E1 -12714.724,E2 -12714.724} C_VEL
LIN {X 0,Y 370.5,Z 858.386,A -85,B 0,C 180,E1 -12718.311,E2 -12718.311} C_VEL
LIN {X 0,Y 371.651,Z 845.367,A -85,B 0,C 180,E1 -12722.292,E2 -12722.292} C_VEL
LIN {X 0,Y 372.758,Z 834.036,A -85,B 0,C 180,E1 -12725.833,E2 -12725.833} C_VEL
LIN {X 0,Y 373.117,Z 830.15,A -85,B 0,C 180,E1 -12727.069,E2 -12727.069} C_VEL
LIN {X 0,Y 372.717,Z 825.973,A -85,B 0,C 180,E1 -12728.483,E2 -12728.483} C_VEL
LIN {X 0,Y 370.919,Z 816.48,A -85,B 0,C 180,E1 -12731.92,E2 -12731.92} C_VEL
LIN {X 0,Y 368.987,Z 807.206,A -85,B 0,C 180,E1 -12735.522,E2 -12735.522} C_VEL
LIN {X 0,Y 368.86,Z 806.542,A -85,B 0,C 180,E1 -12735.832,E2 -12735.832} C_VEL
LIN {X 0,Y 368.889,Z 806.535,A -85,B 0,C 180,E1 -12739.649,E2 -12739.649} C_VEL
LIN {X 0,Y 368.897,Z 806.533,A -85,B 0,C 180,E1 -12743.147,E2 -12743.147} C_VEL
LIN {X 0,Y 368.9,Z 806.535,A -85,B 0,C 180,E1 -12746.462,E2 -12746.462} C_VEL
LIN {X 0,Y 368.902,Z 806.534,A -85,B 0,C 180,E1 -12749.044,E2 -12749.044} C_VEL
LIN {X 0,Y 368.912,Z 806.531,A -85,B 0,C 180,E1 -12751.558,E2 -12751.558} C_VEL
LIN {X 0,Y 368.922,Z 806.53,A -85,B 0,C 180,E1 -12754.014,E2 -12754.014} C_VEL
LIN {X 0,Y 368.898,Z 806.533,A -85,B 0,C 180,E1 -12757.603,E2 -12757.603} C_VEL
LIN {X 0,Y 368.898,Z 806.537,A -85,B 0,C 180,E1 -12759.855,E2 -12759.855} C_VEL
LIN {X 0,Y 369.613,Z 808.845,A -85,B 0,C 180,E1 -12760.089,E2 -12760.089} C_VEL
LIN {X 0,Y 372.83,Z 815.856,A -85,B 0,C 180,E1 -12760.891,E2 -12760.891} C_VEL
LIN {X 0,Y 376.108,Z 825.076,A -85,B 0,C 180,E1 -12761.975,E2 -12761.975} C_VEL
LIN {X 0,Y 377.168,Z 828.943,A -85,B 0,C 180,E1 -12762.445,E2 -12762.445} C_VEL
LIN {X 0,Y 376.308,Z 839.295,A -85,B 0,C 180,E1 -12763.499,E2 -12763.499} C_VEL
LIN {X 0,Y 375.211,Z 849.629,A -85,B 0,C 180,E1 -12764.798,E2 -12764.798} C_VEL
LIN {X 0,Y 374.004,Z 859.877,A -85,B 0,C 180,E1 -12766.415,E2 -12766.415} C_VEL
LIN {X 0,Y 372.946,Z 867.918,A -85,B 0,C 180,E1 -12768.036,E2 -12768.036} C_VEL
LIN {X 0,Y 371.91,Z 875.345,A -85,B 0,C 180,E1 -12769.9,E2 -12769.9} C_VEL
LIN {X 0,Y 371.006,Z 881.102,A -85,B 0,C 180,E1 -12771.832,E2 -12771.832} C_VEL
LIN {X 0,Y 370.166,Z 884.689,A -85,B 0,C 180,E1 -12773.459,E2 -12773.459} C_VEL
LIN {X 0,Y 369.979,Z 886.57,A -85,B 0,C 180,E1 -12774.55,E2 -12774.55} C_VEL
LIN {X 0,Y 369.539,Z 888.818,A -85,B 0,C 180,E1 -12776.729,E2 -12776.729} C_VEL
LIN {X 0,Y 369.338,Z 889.46,A -85,B 0,C 180,E1 -12777.819,E2 -12777.819} C_VEL
LIN {X 0,Y 369.107,Z 889.593,A -85,B 0,C 180,E1 -12778.909,E2 -12778.909} C_VEL
LIN {X 0,Y 369.006,Z 889.318,A -85,B 0,C 180,E1 -12780,E2 -12780} C_VEL
LIN {X 0,Y 369.005,Z 888.643,A -85,B 0,C 180,E1 -12781.091,E2 -12781.091} C_VEL
LIN {X 0,Y 368.848,Z 885.964,A -85,B 0,C 180,E1 -12783.277,E2 -12783.277} C_VEL
LIN {X 0,Y 369.135,Z 882.834,A -85,B 0,C 180,E1 -12784.915,E2 -12784.915} C_VEL
LIN {X 0,Y 369.439,Z 880.246,A -85,B 0,C 180,E1 -12786.006,E2 -12786.006} C_VEL
LIN {X 0,Y 369.717,Z 874.32,A -85,B 0,C 180,E1 -12787.922,E2 -12787.922} C_VEL
LIN {X 0,Y 370.03,Z 869.335,A -85,B 0,C 180,E1 -12789.236,E2 -12789.236} C_VEL
LIN {X 0,Y 370.607,Z 861.453,A -85,B 0,C 180,E1 -12790.932,E2 -12790.932} C_VEL
LIN {X 0,Y 371.052,Z 853.574,A -85,B 0,C 180,E1 -12792.303,E2 -12792.303} C_VEL
LIN {X 0,Y 371.653,Z 845.207,A -85,B 0,C 180,E1 -12793.534,E2 -12793.534} C_VEL
LIN {X 0,Y 372.16,Z 837.579,A -85,B 0,C 180,E1 -12794.49,E2 -12794.49} C_VEL
LIN {X 0,Y 372.815,Z 827.443,A -85,B 0,C 180,E1 -12795.575,E2 -12795.575} C_VEL
LIN {X 0,Y 373.001,Z 822.073,A -85,B 0,C 180,E1 -12796.065,E2 -12796.065} C_VEL
LIN {X 0,Y 369.837,Z 809.909,A -85,B 0,C 180,E1 -12797.13,E2 -12797.13} C_VEL
LIN {X 0,Y 368.936,Z 806.532,A -85,B 0,C 180,E1 -12797.424,E2 -12797.424} C_VEL
LIN {X 0,Y 368.892,Z 806.527,A -85,B 0,C 180,E1 -12801.222,E2 -12801.222} C_VEL
LIN {X 0,Y 368.913,Z 806.532,A -85,B 0,C 180,E1 -12803.873,E2 -12803.873} C_VEL
LIN {X 0,Y 368.862,Z 806.529,A -85,B 0,C 180,E1 -12807.212,E2 -12807.212} C_VEL
LIN {X 0,Y 368.899,Z 806.532,A -85,B 0,C 180,E1 -12809.692,E2 -12809.692} C_VEL
LIN {X 0,Y 368.903,Z 806.521,A -85,B 0,C 180,E1 -12813.042,E2 -12813.042} C_VEL
LIN {X 0,Y 368.917,Z 806.527,A -85,B 0,C 180,E1 -12816.197,E2 -12816.197} C_VEL
LIN {X 0,Y 368.879,Z 806.53,A -85,B 0,C 180,E1 -12818.956,E2 -12818.956} C_VEL
LIN {X 0,Y 368.877,Z 806.532,A -85,B 0,C 180,E1 -12822.007,E2 -12822.007} C_VEL
LIN {X 0,Y 368.885,Z 806.532,A -85,B 0,C 180,E1 -12825.175,E2 -12825.175} C_VEL
LIN {X 0,Y 368.877,Z 806.539,A -85,B 0,C 180,E1 -12828.175,E2 -12828.175} C_VEL
LIN {X 0,Y 368.883,Z 806.533,A -85,B 0,C 180,E1 -12831.365,E2 -12831.365} C_VEL
LIN {X 0,Y 368.943,Z 806.525,A -85,B 0,C 180,E1 -12835.145,E2 -12835.145} C_VEL
LIN {X 0,Y 368.936,Z 806.523,A -85,B 0,C 180,E1 -12839.045,E2 -12839.045} C_VEL
LIN {X 0,Y 368.969,Z 806.518,A -85,B 0,C 180,E1 -12842.795,E2 -12842.795} C_VEL
LIN {X 0,Y 368.95,Z 806.518,A -85,B 0,C 180,E1 -12846.112,E2 -12846.112} C_VEL
LIN {X 0,Y 368.943,Z 806.531,A -85,B 0,C 180,E1 -12849.946,E2 -12849.946} C_VEL
LIN {X 0,Y 368.976,Z 806.529,A -85,B 0,C 180,E1 -12851.18,E2 -12851.18} C_VEL
LIN {X 0,Y 372.775,Z 817.972,A -85,B 0,C 180,E1 -12852.142,E2 -12852.142} C_VEL
LIN {X 0,Y 375.345,Z 827.005,A -85,B 0,C 180,E1 -12853.035,E2 -12853.035} C_VEL
LIN {X 0,Y 374.532,Z 837.701,A -85,B 0,C 180,E1 -12854.07,E2 -12854.07} C_VEL
LIN {X 0,Y 373.68,Z 847.801,A -85,B 0,C 180,E1 -12855.29,E2 -12855.29} C_VEL
LIN {X 0,Y 372.843,Z 856.841,A -85,B 0,C 180,E1 -12856.648,E2 -12856.648} C_VEL
LIN {X 0,Y 371.851,Z 865.613,A -85,B 0,C 180,E1 -12858.275,E2 -12858.275} C_VEL
LIN {X 0,Y 371.093,Z 873.005,A -85,B 0,C 180,E1 -12860.002,E2 -12860.002} C_VEL
LIN {X 0,Y 370.472,Z 879.04,A -85,B 0,C 180,E1 -12861.818,E2 -12861.818} C_VEL
LIN {X 0,Y 369.733,Z 883.303,A -85,B 0,C 180,E1 -12863.449,E2 -12863.449} C_VEL
LIN {X 0,Y 369.508,Z 885.529,A -85,B 0,C 180,E1 -12864.541,E2 -12864.541} C_VEL
LIN {X 0,Y 369.285,Z 887.347,A -85,B 0,C 180,E1 -12865.632,E2 -12865.632} C_VEL
LIN {X 0,Y 369.253,Z 888.698,A -85,B 0,C 180,E1 -12866.725,E2 -12866.725} C_VEL
LIN {X 0,Y 369.101,Z 890.266,A -85,B 0,C 180,E1 -12868.907,E2 -12868.907} C_VEL
LIN {X 0,Y 369.069,Z 890.497,A -85,B 0,C 180,E1 -12869.998,E2 -12869.998} C_VEL
LIN {X 0,Y 369.187,Z 889.739,A -85,B 0,C 180,E1 -12872.18,E2 -12872.18} C_VEL
LIN {X 0,Y 369.274,Z 887.501,A -85,B 0,C 180,E1 -12874.364,E2 -12874.364} C_VEL
LIN {X 0,Y 369.62,Z 884.697,A -85,B 0,C 180,E1 -12876.001,E2 -12876.001} C_VEL
LIN {X 0,Y 370.285,Z 880.862,A -85,B 0,C 180,E1 -12877.633,E2 -12877.633} C_VEL
LIN {X 0,Y 370.896,Z 875.259,A -85,B 0,C 180,E1 -12879.47,E2 -12879.47} C_VEL
LIN {X 0,Y 371.539,Z 868.585,A -85,B 0,C 180,E1 -12881.178,E2 -12881.178} C_VEL
LIN {X 0,Y 372.462,Z 860.564,A -85,B 0,C 180,E1 -12882.807,E2 -12882.807} C_VEL
LIN {X 0,Y 373.269,Z 852.347,A -85,B 0,C 180,E1 -12884.166,E2 -12884.166} C_VEL
LIN {X 0,Y 374.143,Z 842.175,A -85,B 0,C 180,E1 -12885.524,E2 -12885.524} C_VEL
LIN {X 0,Y 375.111,Z 831.807,A -85,B 0,C 180,E1 -12886.625,E2 -12886.625} C_VEL
LIN {X 0,Y 375.384,Z 826.934,A -85,B 0,C 180,E1 -12887.071,E2 -12887.071} C_VEL
LIN {X 0,Y 372.173,Z 816.207,A -85,B 0,C 180,E1 -12888.126,E2 -12888.126} C_VEL
LIN {X 0,Y 368.993,Z 806.52,A -85,B 0,C 180,E1 -12888.926,E2 -12888.926} C_VEL
LIN {X 0,Y 368.923,Z 806.527,A -85,B 0,C 180,E1 -12892.738,E2 -12892.738} C_VEL
LIN {X 0,Y 368.977,Z 806.523,A -85,B 0,C 180,E1 -12896.463,E2 -12896.463} C_VEL
LIN {X 0,Y 368.951,Z 806.524,A -85,B 0,C 180,E1 -12897.481,E2 -12897.481} C_VEL
LIN {X 0,Y 368.262,Z 806.613,A -85,B 0,C 180,E1 -12898.392,E2 -12898.392} C_VEL
LIN {X 0,Y 365.366,Z 806.976,A -85,B 0,C 180,E1 -12899.873,E2 -12899.873} C_VEL
LIN {X 0,Y 362.928,Z 807.278,A -85,B 0,C 180,E1 -12901.07,E2 -12901.07} C_VEL
LIN {X 0,Y 361.893,Z 807.409,A -85,B 0,C 180,E1 -12901.997,E2 -12901.997} C_VEL
LIN {X 0,Y 361.814,Z 807.413,A -85,B 0,C 180,E1 -12902.311,E2 -12902.311} C_VEL
LIN {X 0,Y 361.861,Z 807.41,A -85,B 0,C 180,E1 -12905.634,E2 -12905.634} C_VEL
LIN {X 0,Y 361.866,Z 807.407,A -85,B 0,C 180,E1 -12909.026,E2 -12909.026} C_VEL
LIN {X 0,Y 361.882,Z 807.409,A -85,B 0,C 180,E1 -12912.44,E2 -12912.44} C_VEL
LIN {X 0,Y 361.92,Z 807.402,A -85,B 0,C 180,E1 -12915.926,E2 -12915.926} C_VEL
LIN {X 0,Y 361.894,Z 807.404,A -85,B 0,C 180,E1 -12919.23,E2 -12919.23} C_VEL
LIN {X 0,Y 361.865,Z 807.409,A -85,B 0,C 180,E1 -12922.981,E2 -12922.981} C_VEL
LIN {X 0,Y 361.845,Z 807.41,A -85,B 0,C 180,E1 -12926.629,E2 -12926.629} C_VEL
LIN {X 0,Y 361.863,Z 807.402,A -85,B 0,C 180,E1 -12929.671,E2 -12929.671} C_VEL
LIN {X 0,Y 361.94,Z 807.395,A -85,B 0,C 180,E1 -12933.474,E2 -12933.474} C_VEL
LIN {X 0,Y 361.875,Z 807.408,A -85,B 0,C 180,E1 -12937.144,E2 -12937.144} C_VEL
LIN {X 0,Y 361.891,Z 807.404,A -85,B 0,C 180,E1 -12940.722,E2 -12940.722} C_VEL
LIN {X 0,Y 361.917,Z 807.401,A -85,B 0,C 180,E1 -12943.065,E2 -12943.065} C_VEL
LIN {X 0,Y 361.984,Z 807.391,A -85,B 0,C 180,E1 -12946.527,E2 -12946.527} C_VEL
LIN {X 0,Y 362.02,Z 807.384,A -85,B 0,C 180,E1 -12949.938,E2 -12949.938} C_VEL
LIN {X 0,Y 362.144,Z 807.379,A -85,B 0,C 180,E1 -12953.313,E2 -12953.313} C_VEL
LIN {X 0,Y 362.265,Z 807.361,A -85,B 0,C 180,E1 -12957.776,E2 -12957.776} C_VEL
LIN {X 0,Y 362.41,Z 807.343,A -85,B 0,C 180,E1 -12960,E2 -12960} C_VEL
LIN {X 0,Y 362.263,Z 807.361,A -85,B 0,C 180,E1 -12962.224,E2 -12962.224} C_VEL
LIN {X 0,Y 362.128,Z 807.373,A -85,B 0,C 180,E1 -12966.687,E2 -12966.687} C_VEL
LIN {X 0,Y 362.018,Z 807.391,A -85,B 0,C 180,E1 -12970.062,E2 -12970.062} C_VEL
LIN {X 0,Y 361.982,Z 807.396,A -85,B 0,C 180,E1 -12973.9,E2 -12973.9} C_VEL
LIN {X 0,Y 361.951,Z 807.402,A -85,B 0,C 180,E1 -12977.939,E2 -12977.939} C_VEL
LIN {X 0,Y 361.845,Z 807.414,A -85,B 0,C 180,E1 -12981.656,E2 -12981.656} C_VEL
LIN {X 0,Y 361.862,Z 807.407,A -85,B 0,C 180,E1 -12985.295,E2 -12985.295} C_VEL
LIN {X 0,Y 361.84,Z 807.411,A -85,B 0,C 180,E1 -12989.075,E2 -12989.075} C_VEL
LIN {X 0,Y 361.833,Z 807.413,A -85,B 0,C 180,E1 -12992.946,E2 -12992.946} C_VEL
LIN {X 0,Y 361.849,Z 807.411,A -85,B 0,C 180,E1 -12995.639,E2 -12995.639} C_VEL
LIN {X 0,Y 361.812,Z 807.418,A -85,B 0,C 180,E1 -12999.019,E2 -12999.019} C_VEL
LIN {X 0,Y 361.818,Z 807.412,A -85,B 0,C 180,E1 -13002.832,E2 -13002.832} C_VEL
LIN {X 0,Y 361.856,Z 807.494,A -85,B 0,C 180,E1 -13003.787,E2 -13003.787} C_VEL
LIN {X 0,Y 363.775,Z 816.673,A -85,B 0,C 180,E1 -13007.457,E2 -13007.457} C_VEL
LIN {X 0,Y 365.568,Z 826.108,A -85,B 0,C 180,E1 -13010.972,E2 -13010.972} C_VEL
LIN {X 0,Y 366.198,Z 831.354,A -85,B 0,C 180,E1 -13012.807,E2 -13012.807} C_VEL
LIN {X 0,Y 364.849,Z 844.479,A -85,B 0,C 180,E1 -13017.035,E2 -13017.035} C_VEL
LIN {X 0,Y 363.615,Z 857.464,A -85,B 0,C 180,E1 -13021.108,E2 -13021.108} C_VEL
LIN {X 0,Y 362.849,Z 867.298,A -85,B 0,C 180,E1 -13024.166,E2 -13024.166} C_VEL
LIN {X 0,Y 362.076,Z 878.873,A -85,B 0,C 180,E1 -13027.762,E2 -13027.762} C_VEL
LIN {X 0,Y 361.74,Z 885.593,A -85,B 0,C 180,E1 -13029.867,E2 -13029.867} C_VEL
LIN {X 0,Y 363.685,Z 901.491,A -85,B 0,C 180,E1 -13030.512,E2 -13030.512} C_VEL
LIN {X 0,Y 364.701,Z 915.29,A -85,B 0,C 180,E1 -13031.299,E2 -13031.299} C_VEL
LIN {X 0,Y 365.104,Z 927.586,A -85,B 0,C 180,E1 -13032.209,E2 -13032.209} C_VEL
LIN {X 0,Y 365.387,Z 934.182,A -85,B 0,C 180,E1 -13032.801,E2 -13032.801} C_VEL
LIN {X 0,Y 364.281,Z 944.924,A -85,B 0,C 180,E1 -13033.901,E2 -13033.901} C_VEL
LIN {X 0,Y 363.3,Z 954.785,A -85,B 0,C 180,E1 -13035.15,E2 -13035.15} C_VEL
LIN {X 0,Y 362.76,Z 961.036,A -85,B 0,C 180,E1 -13036.084,E2 -13036.084} C_VEL
LIN {X 0,Y 361.94,Z 969.897,A -85,B 0,C 180,E1 -13037.669,E2 -13037.669} C_VEL
LIN {X 0,Y 361.345,Z 977.535,A -85,B 0,C 180,E1 -13039.354,E2 -13039.354} C_VEL
LIN {X 0,Y 361.087,Z 983.712,A -85,B 0,C 180,E1 -13041.044,E2 -13041.044} C_VEL
LIN {X 0,Y 360.987,Z 988.618,A -85,B 0,C 180,E1 -13042.733,E2 -13042.733} C_VEL
LIN {X 0,Y 361.036,Z 992.391,A -85,B 0,C 180,E1 -13044.417,E2 -13044.417} C_VEL
LIN {X 0,Y 361.179,Z 994.355,A -85,B 0,C 180,E1 -13045.538,E2 -13045.538} C_VEL
LIN {X 0,Y 361.217,Z 995.818,A -85,B 0,C 180,E1 -13046.656,E2 -13046.656} C_VEL
LIN {X 0,Y 361.25,Z 996.86,A -85,B 0,C 180,E1 -13047.772,E2 -13047.772} C_VEL
LIN {X 0,Y 361.3,Z 997.5,A -85,B 0,C 180,E1 -13048.887,E2 -13048.887} C_VEL
LIN {X 0,Y 361.341,Z 997.729,A -85,B 0,C 180,E1 -13050.002,E2 -13050.002} C_VEL
LIN {X 0,Y 361.3,Z 997.495,A -85,B 0,C 180,E1 -13051.117,E2 -13051.117} C_VEL
LIN {X 0,Y 361.25,Z 996.852,A -85,B 0,C 180,E1 -13052.232,E2 -13052.232} C_VEL
LIN {X 0,Y 361.218,Z 995.805,A -85,B 0,C 180,E1 -13053.348,E2 -13053.348} C_VEL
LIN {X 0,Y 361.18,Z 994.337,A -85,B 0,C 180,E1 -13054.466,E2 -13054.466} C_VEL
LIN {X 0,Y 361.028,Z 991.251,A -85,B 0,C 180,E1 -13056.148,E2 -13056.148} C_VEL
LIN {X 0,Y 361.013,Z 987.103,A -85,B 0,C 180,E1 -13057.834,E2 -13057.834} C_VEL
LIN {X 0,Y 361.206,Z 980.756,A -85,B 0,C 180,E1 -13059.804,E2 -13059.804} C_VEL
LIN {X 0,Y 361.602,Z 973.866,A -85,B 0,C 180,E1 -13061.493,E2 -13061.493} C_VEL
LIN {X 0,Y 362.345,Z 965.377,A -85,B 0,C 180,E1 -13063.175,E2 -13063.175} C_VEL
LIN {X 0,Y 363.176,Z 956.297,A -85,B 0,C 180,E1 -13064.63,E2 -13064.63} C_VEL
LIN {X 0,Y 364.102,Z 946.009,A -85,B 0,C 180,E1 -13065.967,E2 -13065.967} C_VEL
LIN {X 0,Y 365.414,Z 934.059,A -85,B 0,C 180,E1 -13067.202,E2 -13067.202} C_VEL
LIN {X 0,Y 364.929,Z 921.433,A -85,B 0,C 180,E1 -13068.269,E2 -13068.269} C_VEL
LIN {X 0,Y 364.472,Z 906.475,A -85,B 0,C 180,E1 -13069.429,E2 -13069.429} C_VEL
LIN {X 0,Y 363.823,Z 896.071,A -85,B 0,C 180,E1 -13070.128,E2 -13070.128} C_VEL
LIN {X 0,Y 362.07,Z 885.126,A -85,B 0,C 180,E1 -13070.821,E2 -13070.821} C_VEL
LIN {X 0,Y 361.863,Z 882.949,A -85,B 0,C 180,E1 -13070.962,E2 -13070.962} C_VEL
LIN {X 0,Y 362.715,Z 869.222,A -85,B 0,C 180,E1 -13075.233,E2 -13075.233} C_VEL
LIN {X 0,Y 363.595,Z 857.4,A -85,B 0,C 180,E1 -13078.898,E2 -13078.898} C_VEL
LIN {X 0,Y 364.842,Z 844.428,A -85,B 0,C 180,E1 -13082.971,E2 -13082.971} C_VEL
LIN {X 0,Y 366.078,Z 832.305,A -85,B 0,C 180,E1 -13086.867,E2 -13086.867} C_VEL
LIN {X 0,Y 365.986,Z 828.754,A -85,B 0,C 180,E1 -13088.064,E2 -13088.064} C_VEL
LIN {X 0,Y 364.414,Z 820.096,A -85,B 0,C 180,E1 -13091.223,E2 -13091.223} C_VEL
LIN {X 0,Y 362.845,Z 812.354,A -85,B 0,C 180,E1 -13094.221,E2 -13094.221} C_VEL
LIN {X 0,Y 361.813,Z 807.418,A -85,B 0,C 180,E1 -13096.302,E2 -13096.302} C_VEL
LIN {X 0,Y 361.816,Z 807.417,A -85,B 0,C 180,E1 -13100.134,E2 -13100.134} C_VEL
LIN {X 0,Y 361.863,Z 807.41,A -85,B 0,C 180,E1 -13102.981,E2 -13102.981} C_VEL
LIN {X 0,Y 361.863,Z 807.411,A -85,B 0,C 180,E1 -13106.632,E2 -13106.632} C_VEL
LIN {X 0,Y 361.853,Z 807.41,A -85,B 0,C 180,E1 -13109.67,E2 -13109.67} C_VEL
LIN {X 0,Y 361.858,Z 807.41,A -85,B 0,C 180,E1 -13113.467,E2 -13113.467} C_VEL
LIN {X 0,Y 361.864,Z 807.409,A -85,B 0,C 180,E1 -13117.143,E2 -13117.143} C_VEL
LIN {X 0,Y 361.884,Z 807.521,A -85,B 0,C 180,E1 -13119.171,E2 -13119.171} C_VEL
LIN {X 0,Y 362.602,Z 809.78,A -85,B 0,C 180,E1 -13119.407,E2 -13119.407} C_VEL
LIN {X 0,Y 366.621,Z 818.379,A -85,B 0,C 180,E1 -13120.469,E2 -13120.469} C_VEL
LIN {X 0,Y 370.08,Z 828.413,A -85,B 0,C 180,E1 -13121.721,E2 -13121.721} C_VEL
LIN {X 0,Y 370.853,Z 831.549,A -85,B 0,C 180,E1 -13122.109,E2 -13122.109} C_VEL
LIN {X 0,Y 369.64,Z 843.665,A -85,B 0,C 180,E1 -13123.429,E2 -13123.429} C_VEL
LIN {X 0,Y 368.656,Z 851.815,A -85,B 0,C 180,E1 -13124.52,E2 -13124.52} C_VEL
LIN {X 0,Y 367.57,Z 860.339,A -85,B 0,C 180,E1 -13125.89,E2 -13125.89} C_VEL
LIN {X 0,Y 366.545,Z 867.27,A -85,B 0,C 180,E1 -13127.262,E2 -13127.262} C_VEL
LIN {X 0,Y 365.793,Z 872.524,A -85,B 0,C 180,E1 -13128.488,E2 -13128.488} C_VEL
LIN {X 0,Y 364.897,Z 877.939,A -85,B 0,C 180,E1 -13130.018,E2 -13130.018} C_VEL
LIN {X 0,Y 364.158,Z 882.645,A -85,B 0,C 180,E1 -13131.678,E2 -13131.678} C_VEL
LIN {X 0,Y 363.261,Z 886.124,A -85,B 0,C 180,E1 -13133.334,E2 -13133.334} C_VEL
LIN {X 0,Y 363.07,Z 887.932,A -85,B 0,C 180,E1 -13134.446,E2 -13134.446} C_VEL
LIN {X 0,Y 362.786,Z 889.212,A -85,B 0,C 180,E1 -13135.556,E2 -13135.556} C_VEL
LIN {X 0,Y 362.352,Z 890.665,A -85,B 0,C 180,E1 -13137.777,E2 -13137.777} C_VEL
LIN {X 0,Y 361.994,Z 890.429,A -85,B 0,C 180,E1 -13140,E2 -13140} C_VEL
LIN {X 0,Y 361.988,Z 889.69,A -85,B 0,C 180,E1 -13141.113,E2 -13141.113} C_VEL
LIN {X 0,Y 361.82,Z 886.888,A -85,B 0,C 180,E1 -13143.341,E2 -13143.341} C_VEL
LIN {X 0,Y 361.944,Z 884.947,A -85,B 0,C 180,E1 -13144.455,E2 -13144.455} C_VEL
LIN {X 0,Y 362.41,Z 881.016,A -85,B 0,C 180,E1 -13146.123,E2 -13146.123} C_VEL
LIN {X 0,Y 362.668,Z 875.964,A -85,B 0,C 180,E1 -13147.796,E2 -13147.796} C_VEL
LIN {X 0,Y 363.037,Z 869.862,A -85,B 0,C 180,E1 -13149.415,E2 -13149.415} C_VEL
LIN {X 0,Y 363.636,Z 861.885,A -85,B 0,C 180,E1 -13151.144,E2 -13151.144} C_VEL
LIN {X 0,Y 364.113,Z 853.846,A -85,B 0,C 180,E1 -13152.541,E2 -13152.541} C_VEL
LIN {X 0,Y 364.669,Z 846.351,A -85,B 0,C 180,E1 -13153.656,E2 -13153.656} C_VEL
LIN {X 0,Y 365.202,Z 838.741,A -85,B 0,C 180,E1 -13154.63,E2 -13154.63} C_VEL
LIN {X 0,Y 365.852,Z 828.497,A -85,B 0,C 180,E1 -13155.75,E2 -13155.75} C_VEL
LIN {X 0,Y 366.013,Z 823.255,A -85,B 0,C 180,E1 -13156.241,E2 -13156.241} C_VEL
LIN {X 0,Y 362.988,Z 811.573,A -85,B 0,C 180,E1 -13157.293,E2 -13157.293} C_VEL
LIN {X 0,Y 361.88,Z 807.41,A -85,B 0,C 180,E1 -13157.651,E2 -13157.651} C_VEL
LIN {X 0,Y 361.832,Z 807.406,A -85,B 0,C 180,E1 -13161.657,E2 -13161.657} C_VEL
LIN {X 0,Y 361.858,Z 807.409,A -85,B 0,C 180,E1 -13165.295,E2 -13165.295} C_VEL
LIN {X 0,Y 361.862,Z 807.403,A -85,B 0,C 180,E1 -13169.073,E2 -13169.073} C_VEL
LIN {X 0,Y 361.854,Z 807.398,A -85,B 0,C 180,E1 -13172.944,E2 -13172.944} C_VEL
LIN {X 0,Y 361.87,Z 807.408,A -85,B 0,C 180,E1 -13175.637,E2 -13175.637} C_VEL
LIN {X 0,Y 361.831,Z 807.408,A -85,B 0,C 180,E1 -13179.017,E2 -13179.017} C_VEL
LIN {X 0,Y 361.839,Z 807.407,A -85,B 0,C 180,E1 -13182.829,E2 -13182.829} C_VEL
LIN {X 0,Y 361.824,Z 807.413,A -85,B 0,C 180,E1 -13185.946,E2 -13185.946} C_VEL
LIN {X 0,Y 361.819,Z 807.412,A -85,B 0,C 180,E1 -13189.248,E2 -13189.248} C_VEL
LIN {X 0,Y 361.871,Z 807.403,A -85,B 0,C 180,E1 -13192.981,E2 -13192.981} C_VEL
LIN {X 0,Y 361.866,Z 807.408,A -85,B 0,C 180,E1 -13196.63,E2 -13196.63} C_VEL
LIN {X 0,Y 361.88,Z 807.402,A -85,B 0,C 180,E1 -13199.671,E2 -13199.671} C_VEL
LIN {X 0,Y 361.96,Z 807.39,A -85,B 0,C 180,E1 -13203.474,E2 -13203.474} C_VEL
LIN {X 0,Y 361.898,Z 807.404,A -85,B 0,C 180,E1 -13207.143,E2 -13207.143} C_VEL
LIN {X 0,Y 361.901,Z 807.411,A -85,B 0,C 180,E1 -13210.784,E2 -13210.784} C_VEL
LIN {X 0,Y 365.82,Z 819.053,A -85,B 0,C 180,E1 -13211.791,E2 -13211.791} C_VEL
LIN {X 0,Y 368.537,Z 828.469,A -85,B 0,C 180,E1 -13212.75,E2 -13212.75} C_VEL
LIN {X 0,Y 368.264,Z 833.377,A -85,B 0,C 180,E1 -13213.214,E2 -13213.214} C_VEL
LIN {X 0,Y 367.37,Z 843.486,A -85,B 0,C 180,E1 -13214.321,E2 -13214.321} C_VEL
LIN {X 0,Y 366.545,Z 852.673,A -85,B 0,C 180,E1 -13215.565,E2 -13215.565} C_VEL
LIN {X 0,Y 365.665,Z 861.042,A -85,B 0,C 180,E1 -13216.946,E2 -13216.946} C_VEL
LIN {X 0,Y 364.703,Z 869.158,A -85,B 0,C 180,E1 -13218.606,E2 -13218.606} C_VEL
LIN {X 0,Y 363.936,Z 875.894,A -85,B 0,C 180,E1 -13220.333,E2 -13220.333} C_VEL
LIN {X 0,Y 363.311,Z 881.632,A -85,B 0,C 180,E1 -13222.216,E2 -13222.216} C_VEL
LIN {X 0,Y 362.645,Z 885.526,A -85,B 0,C 180,E1 -13223.879,E2 -13223.879} C_VEL
LIN {X 0,Y 362.281,Z 888.379,A -85,B 0,C 180,E1 -13225.548,E2 -13225.548} C_VEL
LIN {X 0,Y 362.262,Z 889.726,A -85,B 0,C 180,E1 -13226.662,E2 -13226.662} C_VEL
LIN {X 0,Y 362.08,Z 891.297,A -85,B 0,C 180,E1 -13228.886,E2 -13228.886} C_VEL
LIN {X 0,Y 362.045,Z 891.528,A -85,B 0,C 180,E1 -13229.998,E2 -13229.998} C_VEL
LIN {X 0,Y 362.175,Z 890.769,A -85,B 0,C 180,E1 -13232.222,E2 -13232.222} C_VEL
LIN {X 0,Y 362.27,Z 888.532,A -85,B 0,C 180,E1 -13234.449,E2 -13234.449} C_VEL
LIN {X 0,Y 362.634,Z 885.727,A -85,B 0,C 180,E1 -13236.117,E2 -13236.117} C_VEL
LIN {X 0,Y 363.327,Z 881.891,A -85,B 0,C 180,E1 -13237.78,E2 -13237.78} C_VEL
LIN {X 0,Y 363.969,Z 876.279,A -85,B 0,C 180,E1 -13239.655,E2 -13239.655} C_VEL
LIN {X 0,Y 364.649,Z 869.614,A -85,B 0,C 180,E1 -13241.392,E2 -13241.392} C_VEL
LIN {X 0,Y 365.617,Z 861.593,A -85,B 0,C 180,E1 -13243.051,E2 -13243.051} C_VEL
LIN {X 0,Y 366.462,Z 853.375,A -85,B 0,C 180,E1 -13244.435,E2 -13244.435} C_VEL
LIN {X 0,Y 367.394,Z 843.2,A -85,B 0,C 180,E1 -13245.816,E2 -13245.816} C_VEL
LIN {X 0,Y 368.39,Z 832.833,A -85,B 0,C 180,E1 -13246.937,E2 -13246.937} C_VEL
LIN {X 0,Y 368.681,Z 828.833,A -85,B 0,C 180,E1 -13247.31,E2 -13247.31} C_VEL
LIN {X 0,Y 365.731,Z 818.813,A -85,B 0,C 180,E1 -13248.336,E2 -13248.336} C_VEL
LIN {X 0,Y 361.926,Z 807.4,A -85,B 0,C 180,E1 -13249.347,E2 -13249.347} C_VEL
LIN {X 0,Y 361.887,Z 807.404,A -85,B 0,C 180,E1 -13252.853,E2 -13252.853} C_VEL
LIN {X 0,Y 361.938,Z 807.399,A -85,B 0,C 180,E1 -13256.72,E2 -13256.72} C_VEL
LIN {X 0,Y 361.869,Z 807.41,A -85,B 0,C 180,E1 -13260.326,E2 -13260.326} C_VEL
LIN {X 0,Y 361.814,Z 807.413,A -85,B 0,C 180,E1 -13262.311,E2 -13262.311} C_VEL
LIN {X 0,Y 361.157,Z 807.497,A -85,B 0,C 180,E1 -13263.241,E2 -13263.241} C_VEL
LIN {X 0,Y 358.294,Z 807.854,A -85,B 0,C 180,E1 -13264.753,E2 -13264.753} C_VEL
LIN {X 0,Y 355.876,Z 808.159,A -85,B 0,C 180,E1 -13265.976,E2 -13265.976} C_VEL
LIN {X 0,Y 354.856,Z 808.282,A -85,B 0,C 180,E1 -13266.923,E2 -13266.923} C_VEL
LIN {X 0,Y 354.783,Z 808.29,A -85,B 0,C 180,E1 -13267.244,E2 -13267.244} C_VEL
LIN {X 0,Y 354.849,Z 808.282,A -85,B 0,C 180,E1 -13270.809,E2 -13270.809} C_VEL
LIN {X 0,Y 354.877,Z 808.282,A -85,B 0,C 180,E1 -13274.525,E2 -13274.525} C_VEL
LIN {X 0,Y 354.829,Z 808.279,A -85,B 0,C 180,E1 -13277.667,E2 -13277.667} C_VEL
LIN {X 0,Y 354.841,Z 808.281,A -85,B 0,C 180,E1 -13280.669,E2 -13280.669} C_VEL
LIN {X 0,Y 354.81,Z 808.289,A -85,B 0,C 180,E1 -13284.299,E2 -13284.299} C_VEL
LIN {X 0,Y 354.774,Z 808.29,A -85,B 0,C 180,E1 -13287.665,E2 -13287.665} C_VEL
LIN {X 0,Y 354.855,Z 808.279,A -85,B 0,C 180,E1 -13290.62,E2 -13290.62} C_VEL
LIN {X 0,Y 354.885,Z 808.274,A -85,B 0,C 180,E1 -13294.171,E2 -13294.171} C_VEL
LIN {X 0,Y 354.819,Z 808.283,A -85,B 0,C 180,E1 -13297.893,E2 -13297.893} C_VEL
LIN {X 0,Y 354.906,Z 808.273,A -85,B 0,C 180,E1 -13301.891,E2 -13301.891} C_VEL
LIN {X 0,Y 354.927,Z 808.269,A -85,B 0,C 180,E1 -13305.98,E2 -13305.98} C_VEL
LIN {X 0,Y 354.967,Z 808.264,A -85,B 0,C 180,E1 -13309.735,E2 -13309.735} C_VEL
LIN {X 0,Y 355.108,Z 808.254,A -85,B 0,C 180,E1 -13313.18,E2 -13313.18} C_VEL
LIN {X 0,Y 355.228,Z 808.237,A -85,B 0,C 180,E1 -13317.732,E2 -13317.732} C_VEL
LIN {X 0,Y 355.38,Z 808.219,A -85,B 0,C 180,E1 -13320,E2 -13320} C_VEL
LIN {X 0,Y 355.227,Z 808.237,A -85,B 0,C 180,E1 -13322.268,E2 -13322.268} C_VEL
LIN {X 0,Y 355.095,Z 808.25,A -85,B 0,C 180,E1 -13326.82,E2 -13326.82} C_VEL
LIN {X 0,Y 354.994,Z 808.263,A -85,B 0,C 180,E1 -13329.113,E2 -13329.113} C_VEL
LIN {X 0,Y 354.909,Z 808.269,A -85,B 0,C 180,E1 -13332.581,E2 -13332.581} C_VEL
LIN {X 0,Y 354.873,Z 808.283,A -85,B 0,C 180,E1 -13336.097,E2 -13336.097} C_VEL
LIN {X 0,Y 354.887,Z 808.28,A -85,B 0,C 180,E1 -13338.473,E2 -13338.473} C_VEL
LIN {X 0,Y 354.799,Z 808.293,A -85,B 0,C 180,E1 -13342.108,E2 -13342.108} C_VEL
LIN {X 0,Y 354.832,Z 808.285,A -85,B 0,C 180,E1 -13344.578,E2 -13344.578} C_VEL
LIN {X 0,Y 354.786,Z 808.293,A -85,B 0,C 180,E1 -13348.387,E2 -13348.387} C_VEL
LIN {X 0,Y 354.772,Z 808.293,A -85,B 0,C 180,E1 -13352.335,E2 -13352.335} C_VEL
LIN {X 0,Y 354.804,Z 808.289,A -85,B 0,C 180,E1 -13355.7,E2 -13355.7} C_VEL
LIN {X 0,Y 354.755,Z 808.296,A -85,B 0,C 180,E1 -13359.414,E2 -13359.414} C_VEL
LIN {X 0,Y 354.81,Z 808.387,A -85,B 0,C 180,E1 -13363.328,E2 -13363.328} C_VEL
LIN {X 0,Y 356.562,Z 816.879,A -85,B 0,C 180,E1 -13366.827,E2 -13366.827} C_VEL
LIN {X 0,Y 358.138,Z 824.922,A -85,B 0,C 180,E1 -13369.936,E2 -13369.936} C_VEL
LIN {X 0,Y 359.167,Z 830.895,A -85,B 0,C 180,E1 -13372.123,E2 -13372.123} C_VEL
LIN {X 0,Y 359.02,Z 834.586,A -85,B 0,C 180,E1 -13373.379,E2 -13373.379} C_VEL
LIN {X 0,Y 357.728,Z 846.304,A -85,B 0,C 180,E1 -13377.224,E2 -13377.224} C_VEL
LIN {X 0,Y 356.546,Z 858.461,A -85,B 0,C 180,E1 -13381.126,E2 -13381.126} C_VEL
LIN {X 0,Y 355.744,Z 868.237,A -85,B 0,C 180,E1 -13384.241,E2 -13384.241} C_VEL
LIN {X 0,Y 354.96,Z 879.729,A -85,B 0,C 180,E1 -13387.905,E2 -13387.905} C_VEL
LIN {X 0,Y 354.699,Z 884.575,A -85,B 0,C 180,E1 -13389.468,E2 -13389.468} C_VEL
LIN {X 0,Y 356.546,Z 899.037,A -85,B 0,C 180,E1 -13390.049,E2 -13390.049} C_VEL
LIN {X 0,Y 357.612,Z 911.756,A -85,B 0,C 180,E1 -13390.757,E2 -13390.757} C_VEL
LIN {X 0,Y 358.019,Z 924.689,A -85,B 0,C 180,E1 -13391.697,E2 -13391.697} C_VEL
LIN {X 0,Y 358.415,Z 934.58,A -85,B 0,C 180,E1 -13392.603,E2 -13392.603} C_VEL
LIN {X 0,Y 357.097,Z 946.251,A -85,B 0,C 180,E1 -13393.862,E2 -13393.862} C_VEL
LIN {X 0,Y 356.172,Z 955.719,A -85,B 0,C 180,E1 -13395.139,E2 -13395.139} C_VEL
LIN {X 0,Y 355.703,Z 960.449,A -85,B 0,C 180,E1 -13395.883,E2 -13395.883} C_VEL
LIN {X 0,Y 354.914,Z 968.842,A -85,B 0,C 180,E1 -13397.421,E2 -13397.421} C_VEL
LIN {X 0,Y 354.305,Z 976.484,A -85,B 0,C 180,E1 -13399.14,E2 -13399.14} C_VEL
LIN {X 0,Y 354.038,Z 982.665,A -85,B 0,C 180,E1 -13400.864,E2 -13400.864} C_VEL
LIN {X 0,Y 353.924,Z 987.722,A -85,B 0,C 180,E1 -13402.644,E2 -13402.644} C_VEL
LIN {X 0,Y 353.973,Z 991.35,A -85,B 0,C 180,E1 -13404.305,E2 -13404.305} C_VEL
LIN {X 0,Y 354.117,Z 993.316,A -85,B 0,C 180,E1 -13405.449,E2 -13405.449} C_VEL
LIN {X 0,Y 354.175,Z 994.782,A -85,B 0,C 180,E1 -13406.589,E2 -13406.589} C_VEL
LIN {X 0,Y 354.212,Z 995.827,A -85,B 0,C 180,E1 -13407.728,E2 -13407.728} C_VEL
LIN {X 0,Y 354.269,Z 996.468,A -85,B 0,C 180,E1 -13408.865,E2 -13408.865} C_VEL
LIN {X 0,Y 354.316,Z 996.698,A -85,B 0,C 180,E1 -13410.002,E2 -13410.002} C_VEL
LIN {X 0,Y 354.269,Z 996.463,A -85,B 0,C 180,E1 -13411.139,E2 -13411.139} C_VEL
LIN {X 0,Y 354.213,Z 995.817,A -85,B 0,C 180,E1 -13412.276,E2 -13412.276} C_VEL
LIN {X 0,Y 354.176,Z 994.768,A -85,B 0,C 180,E1 -13413.415,E2 -13413.415} C_VEL
LIN {X 0,Y 354.118,Z 993.296,A -85,B 0,C 180,E1 -13414.555,E2 -13414.555} C_VEL
LIN {X 0,Y 353.984,Z 989.636,A -85,B 0,C 180,E1 -13416.532,E2 -13416.532} C_VEL
LIN {X 0,Y 353.98,Z 984.395,A -85,B 0,C 180,E1 -13418.566,E2 -13418.566} C_VEL
LIN {X 0,Y 354.213,Z 978.659,A -85,B 0,C 180,E1 -13420.288,E2 -13420.288} C_VEL
LIN {X 0,Y 354.728,Z 971.549,A -85,B 0,C 180,E1 -13422.009,E2 -13422.009} C_VEL
LIN {X 0,Y 355.413,Z 964.329,A -85,B 0,C 180,E1 -13423.437,E2 -13423.437} C_VEL
LIN {X 0,Y 356.21,Z 955.641,A -85,B 0,C 180,E1 -13424.864,E2 -13424.864} C_VEL
LIN {X 0,Y 357.293,Z 944.965,A -85,B 0,C 180,E1 -13426.28,E2 -13426.28} C_VEL
LIN {X 0,Y 358.444,Z 934.452,A -85,B 0,C 180,E1 -13427.4,E2 -13427.4} C_VEL
LIN {X 0,Y 358.07,Z 915.41,A -85,B 0,C 180,E1 -13429.167,E2 -13429.167} C_VEL
LIN {X 0,Y 357.771,Z 901.549,A -85,B 0,C 180,E1 -13430.258,E2 -13430.258} C_VEL
LIN {X 0,Y 355.819,Z 886.929,A -85,B 0,C 180,E1 -13431.277,E2 -13431.277} C_VEL
LIN {X 0,Y 354.884,Z 881.07,A -85,B 0,C 180,E1 -13431.657,E2 -13431.657} C_VEL
LIN {X 0,Y 355.607,Z 870.135,A -85,B 0,C 180,E1 -13435.146,E2 -13435.146} C_VEL
LIN {X 0,Y 356.528,Z 858.389,A -85,B 0,C 180,E1 -13438.88,E2 -13438.88} C_VEL
LIN {X 0,Y 357.73,Z 846.238,A -85,B 0,C 180,E1 -13442.779,E2 -13442.779} C_VEL
LIN {X 0,Y 359.016,Z 834.538,A -85,B 0,C 180,E1 -13446.62,E2 -13446.62} C_VEL
LIN {X 0,Y 359.128,Z 830.869,A -85,B 0,C 180,E1 -13447.878,E2 -13447.878} C_VEL
LIN {X 0,Y 357.652,Z 822.382,A -85,B 0,C 180,E1 -13451.019,E2 -13451.019} C_VEL
LIN {X 0,Y 356.014,Z 814.352,A -85,B 0,C 180,E1 -13454.168,E2 -13454.168} C_VEL
LIN {X 0,Y 354.752,Z 808.297,A -85,B 0,C 180,E1 -13456.744,E2 -13456.744} C_VEL
LIN {X 0,Y 354.791,Z 808.291,A -85,B 0,C 180,E1 -13460.663,E2 -13460.663} C_VEL
LIN {X 0,Y 354.821,Z 808.289,A -85,B 0,C 180,E1 -13464.303,E2 -13464.303} C_VEL
LIN {X 0,Y 354.792,Z 808.289,A -85,B 0,C 180,E1 -13467.667,E2 -13467.667} C_VEL
LIN {X 0,Y 354.794,Z 808.289,A -85,B 0,C 180,E1 -13471.614,E2 -13471.614} C_VEL
LIN {X 0,Y 354.807,Z 808.287,A -85,B 0,C 180,E1 -13475.42,E2 -13475.42} C_VEL
LIN {X 0,Y 354.789,Z 808.307,A -85,B 0,C 180,E1 -13478.403,E2 -13478.403} C_VEL
LIN {X 0,Y 355.59,Z 810.746,A -85,B 0,C 180,E1 -13478.661,E2 -13478.661} C_VEL
LIN {X 0,Y 358.1,Z 815.525,A -85,B 0,C 180,E1 -13479.313,E2 -13479.313} C_VEL
LIN {X 0,Y 361.957,Z 825.112,A -85,B 0,C 180,E1 -13480.553,E2 -13480.553} C_VEL
LIN {X 0,Y 364.545,Z 833.454,A -85,B 0,C 180,E1 -13481.674,E2 -13481.674} C_VEL
LIN {X 0,Y 363.306,Z 845.117,A -85,B 0,C 180,E1 -13482.988,E2 -13482.988} C_VEL
LIN {X 0,Y 362.127,Z 854.084,A -85,B 0,C 180,E1 -13484.234,E2 -13484.234} C_VEL
LIN {X 0,Y 360.976,Z 862.444,A -85,B 0,C 180,E1 -13485.627,E2 -13485.627} C_VEL
LIN {X 0,Y 359.892,Z 869.186,A -85,B 0,C 180,E1 -13487.022,E2 -13487.022} C_VEL
LIN {X 0,Y 359.08,Z 874.312,A -85,B 0,C 180,E1 -13488.27,E2 -13488.27} C_VEL
LIN {X 0,Y 358.113,Z 879.611,A -85,B 0,C 180,E1 -13489.827,E2 -13489.827} C_VEL
LIN {X 0,Y 357.324,Z 884.221,A -85,B 0,C 180,E1 -13491.517,E2 -13491.517} C_VEL
LIN {X 0,Y 356.384,Z 887.579,A -85,B 0,C 180,E1 -13493.205,E2 -13493.205} C_VEL
LIN {X 0,Y 356.153,Z 889.304,A -85,B 0,C 180,E1 -13494.338,E2 -13494.338} C_VEL
LIN {X 0,Y 355.842,Z 890.569,A -85,B 0,C 180,E1 -13495.469,E2 -13495.469} C_VEL
LIN {X 0,Y 355.387,Z 891.87,A -85,B 0,C 180,E1 -13497.733,E2 -13497.733} C_VEL
LIN {X 0,Y 355.132,Z 891.906,A -85,B 0,C 180,E1 -13498.866,E2 -13498.866} C_VEL
LIN {X 0,Y 354.982,Z 891.54,A -85,B 0,C 180,E1 -13500,E2 -13500} C_VEL
LIN {X 0,Y 354.97,Z 890.713,A -85,B 0,C 180,E1 -13501.135,E2 -13501.135} C_VEL
LIN {X 0,Y 354.878,Z 889.46,A -85,B 0,C 180,E1 -13502.27,E2 -13502.27} C_VEL
LIN {X 0,Y 354.915,Z 885.78,A -85,B 0,C 180,E1 -13504.543,E2 -13504.543} C_VEL
LIN {X 0,Y 355.38,Z 881.739,A -85,B 0,C 180,E1 -13506.244,E2 -13506.244} C_VEL
LIN {X 0,Y 355.671,Z 876.574,A -85,B 0,C 180,E1 -13507.951,E2 -13507.951} C_VEL
LIN {X 0,Y 355.981,Z 871.336,A -85,B 0,C 180,E1 -13509.374,E2 -13509.374} C_VEL
LIN {X 0,Y 356.581,Z 863.673,A -85,B 0,C 180,E1 -13511.079,E2 -13511.079} C_VEL
LIN {X 0,Y 357.086,Z 855.797,A -85,B 0,C 180,E1 -13512.503,E2 -13512.503} C_VEL
LIN {X 0,Y 357.681,Z 847.445,A -85,B 0,C 180,E1 -13513.783,E2 -13513.783} C_VEL
LIN {X 0,Y 358.205,Z 839.844,A -85,B 0,C 180,E1 -13514.777,E2 -13514.777} C_VEL
LIN {X 0,Y 358.889,Z 829.671,A -85,B 0,C 180,E1 -13515.912,E2 -13515.912} C_VEL
LIN {X 0,Y 359.028,Z 824.348,A -85,B 0,C 180,E1 -13516.424,E2 -13516.424} C_VEL
LIN {X 0,Y 355.927,Z 812.417,A -85,B 0,C 180,E1 -13517.519,E2 -13517.519} C_VEL
LIN {X 0,Y 354.861,Z 808.282,A -85,B 0,C 180,E1 -13517.854,E2 -13517.854} C_VEL
LIN {X 0,Y 354.797,Z 808.285,A -85,B 0,C 180,E1 -13522.109,E2 -13522.109} C_VEL
LIN {X 0,Y 354.801,Z 808.285,A -85,B 0,C 180,E1 -13525.835,E2 -13525.835} C_VEL
LIN {X 0,Y 354.803,Z 808.288,A -85,B 0,C 180,E1 -13529.683,E2 -13529.683} C_VEL
LIN {X 0,Y 354.793,Z 808.279,A -85,B 0,C 180,E1 -13532.333,E2 -13532.333} C_VEL
LIN {X 0,Y 354.825,Z 808.286,A -85,B 0,C 180,E1 -13535.698,E2 -13535.698} C_VEL
LIN {X 0,Y 354.775,Z 808.288,A -85,B 0,C 180,E1 -13539.412,E2 -13539.412} C_VEL
LIN {X 0,Y 354.792,Z 808.285,A -85,B 0,C 180,E1 -13542.866,E2 -13542.866} C_VEL
LIN {X 0,Y 354.773,Z 808.29,A -85,B 0,C 180,E1 -13546.103,E2 -13546.103} C_VEL
LIN {X 0,Y 354.772,Z 808.29,A -85,B 0,C 180,E1 -13549.175,E2 -13549.175} C_VEL
LIN {X 0,Y 354.807,Z 808.286,A -85,B 0,C 180,E1 -13552.403,E2 -13552.403} C_VEL
LIN {X 0,Y 354.818,Z 808.285,A -85,B 0,C 180,E1 -13554.94,E2 -13554.94} C_VEL
LIN {X 0,Y 354.8,Z 808.285,A -85,B 0,C 180,E1 -13558.404,E2 -13558.404} C_VEL
LIN {X 0,Y 354.853,Z 808.276,A -85,B 0,C 180,E1 -13561.617,E2 -13561.617} C_VEL
LIN {X 0,Y 354.905,Z 808.274,A -85,B 0,C 180,E1 -13564.171,E2 -13564.171} C_VEL
LIN {X 0,Y 354.842,Z 808.284,A -85,B 0,C 180,E1 -13567.893,E2 -13567.893} C_VEL
LIN {X 0,Y 354.892,Z 808.485,A -85,B 0,C 180,E1 -13570.39,E2 -13570.39} C_VEL
LIN {X 0,Y 359.091,Z 820.823,A -85,B 0,C 180,E1 -13571.492,E2 -13571.492} C_VEL
LIN {X 0,Y 361.796,Z 830.222,A -85,B 0,C 180,E1 -13572.486,E2 -13572.486} C_VEL
LIN {X 0,Y 360.941,Z 841.038,A -85,B 0,C 180,E1 -13573.599,E2 -13573.599} C_VEL
LIN {X 0,Y 360.11,Z 849.87,A -85,B 0,C 180,E1 -13574.722,E2 -13574.722} C_VEL
LIN {X 0,Y 359.217,Z 858.905,A -85,B 0,C 180,E1 -13576.131,E2 -13576.131} C_VEL
LIN {X 0,Y 358.105,Z 867.681,A -85,B 0,C 180,E1 -13577.819,E2 -13577.819} C_VEL
LIN {X 0,Y 357.262,Z 875.061,A -85,B 0,C 180,E1 -13579.608,E2 -13579.608} C_VEL
LIN {X 0,Y 356.577,Z 881.105,A -85,B 0,C 180,E1 -13581.497,E2 -13581.497} C_VEL
LIN {X 0,Y 355.781,Z 885.368,A -85,B 0,C 180,E1 -13583.191,E2 -13583.191} C_VEL
LIN {X 0,Y 355.524,Z 887.593,A -85,B 0,C 180,E1 -13584.326,E2 -13584.326} C_VEL
LIN {X 0,Y 355.278,Z 889.411,A -85,B 0,C 180,E1 -13585.46,E2 -13585.46} C_VEL
LIN {X 0,Y 355.268,Z 890.755,A -85,B 0,C 180,E1 -13586.596,E2 -13586.596} C_VEL
LIN {X 0,Y 355.06,Z 892.328,A -85,B 0,C 180,E1 -13588.864,E2 -13588.864} C_VEL
LIN {X 0,Y 355.021,Z 892.559,A -85,B 0,C 180,E1 -13589.998,E2 -13589.998} C_VEL
LIN {X 0,Y 355.161,Z 891.799,A -85,B 0,C 180,E1 -13592.266,E2 -13592.266} C_VEL
LIN {X 0,Y 355.267,Z 889.563,A -85,B 0,C 180,E1 -13594.536,E2 -13594.536} C_VEL
LIN {X 0,Y 355.65,Z 886.758,A -85,B 0,C 180,E1 -13596.237,E2 -13596.237} C_VEL
LIN {X 0,Y 356.372,Z 882.921,A -85,B 0,C 180,E1 -13597.933,E2 -13597.933} C_VEL
LIN {X 0,Y 357.056,Z 877.264,A -85,B 0,C 180,E1 -13599.857,E2 -13599.857} C_VEL
LIN {X 0,Y 357.765,Z 870.643,A -85,B 0,C 180,E1 -13601.614,E2 -13601.614} C_VEL
LIN {X 0,Y 358.782,Z 862.621,A -85,B 0,C 180,E1 -13603.305,E2 -13603.305} C_VEL
LIN {X 0,Y 359.663,Z 854.403,A -85,B 0,C 180,E1 -13604.714,E2 -13604.714} C_VEL
LIN {X 0,Y 360.656,Z 844.225,A -85,B 0,C 180,E1 -13606.12,E2 -13606.12} C_VEL
LIN {X 0,Y 361.521,Z 835.118,A -85,B 0,C 180,E1 -13607.139,E2 -13607.139} C_VEL
LIN {X 0,Y 361.902,Z 831.136,A -85,B 0,C 180,E1 -13607.525,E2 -13607.525} C_VEL
LIN {X 0,Y 359.369,Z 821.669,A -85,B 0,C 180,E1 -13608.53,E2 -13608.53} C_VEL
LIN {X 0,Y 355.955,Z 811.498,A -85,B 0,C 180,E1 -13609.467,E2 -13609.467} C_VEL
LIN {X 0,Y 354.882,Z 808.279,A -85,B 0,C 180,E1 -13609.747,E2 -13609.747} C_VEL
LIN {X 0,Y 354.829,Z 808.285,A -85,B 0,C 180,E1 -13613.334,E2 -13613.334} C_VEL
LIN {X 0,Y 354.884,Z 808.278,A -85,B 0,C 180,E1 -13616.98,E2 -13616.98} C_VEL
LIN {X 0,Y 354.848,Z 808.285,A -85,B 0,C 180,E1 -13619.676,E2 -13619.676} C_VEL
LIN {X 0,Y 354.799,Z 808.291,A -85,B 0,C 180,E1 -13623.7,E2 -13623.7} C_VEL
LIN {X 0,Y 354.783,Z 808.29,A -85,B 0,C 180,E1 -13627.244,E2 -13627.244} C_VEL
LIN {X 0,Y 354.145,Z 808.374,A -85,B 0,C 180,E1 -13628.191,E2 -13628.191} C_VEL
LIN {X 0,Y 351.308,Z 808.727,A -85,B 0,C 180,E1 -13629.733,E2 -13629.733} C_VEL
LIN {X 0,Y 348.888,Z 809.027,A -85,B 0,C 180,E1 -13630.981,E2 -13630.981} C_VEL
LIN {X 0,Y 347.846,Z 809.156,A -85,B 0,C 180,E1 -13631.946,E2 -13631.946} C_VEL
LIN {X 0,Y 347.761,Z 809.162,A -85,B 0,C 180,E1 -13632.273,E2 -13632.273} C_VEL
LIN {X 0,Y 347.821,Z 809.158,A -85,B 0,C 180,E1 -13635.004,E2 -13635.004} C_VEL
LIN {X 0,Y 347.774,Z 809.163,A -85,B 0,C 180,E1 -13638.389,E2 -13638.389} C_VEL
LIN {X 0,Y 347.77,Z 809.159,A -85,B 0,C 180,E1 -13642.008,E2 -13642.008} C_VEL
LIN {X 0,Y 347.731,Z 809.161,A -85,B 0,C 180,E1 -13645.534,E2 -13645.534} C_VEL
LIN {X 0,Y 347.751,Z 809.16,A -85,B 0,C 180,E1 -13649.652,E2 -13649.652} C_VEL
LIN {X 0,Y 347.838,Z 809.159,A -85,B 0,C 180,E1 -13652.743,E2 -13652.743} C_VEL
LIN {X 0,Y 347.773,Z 809.161,A -85,B 0,C 180,E1 -13656.161,E2 -13656.161} C_VEL
LIN {X 0,Y 347.797,Z 809.156,A -85,B 0,C 180,E1 -13659.908,E2 -13659.908} C_VEL
LIN {X 0,Y 347.85,Z 809.153,A -85,B 0,C 180,E1 -13662.358,E2 -13662.358} C_VEL
LIN {X 0,Y 347.881,Z 809.147,A -85,B 0,C 180,E1 -13665.97,E2 -13665.97} C_VEL
LIN {X 0,Y 347.917,Z 809.143,A -85,B 0,C 180,E1 -13669.525,E2 -13669.525} C_VEL
LIN {X 0,Y 348.075,Z 809.129,A -85,B 0,C 180,E1 -13673.042,E2 -13673.042} C_VEL
LIN {X 0,Y 348.19,Z 809.113,A -85,B 0,C 180,E1 -13677.686,E2 -13677.686} C_VEL
LIN {X 0,Y 348.329,Z 809.098,A -85,B 0,C 180,E1 -13680,E2 -13680} C_VEL
LIN {X 0,Y 348.189,Z 809.114,A -85,B 0,C 180,E1 -13682.314,E2 -13682.314} C_VEL
LIN {X 0,Y 348.063,Z 809.126,A -85,B 0,C 180,E1 -13686.958,E2 -13686.958} C_VEL
LIN {X 0,Y 347.948,Z 809.142,A -85,B 0,C 180,E1 -13689.299,E2 -13689.299} C_VEL
LIN {X 0,Y 347.877,Z 809.144,A -85,B 0,C 180,E1 -13692.84,E2 -13692.84} C_VEL
LIN {X 0,Y 347.822,Z 809.159,A -85,B 0,C 180,E1 -13696.432,E2 -13696.432} C_VEL
LIN {X 0,Y 347.836,Z 809.157,A -85,B 0,C 180,E1 -13698.861,E2 -13698.861} C_VEL
LIN {X 0,Y 347.74,Z 809.169,A -85,B 0,C 180,E1 -13702.582,E2 -13702.582} C_VEL
LIN {X 0,Y 347.751,Z 809.165,A -85,B 0,C 180,E1 -13705.113,E2 -13705.113} C_VEL
LIN {X 0,Y 347.722,Z 809.167,A -85,B 0,C 180,E1 -13707.702,E2 -13707.702} C_VEL
LIN {X 0,Y 347.724,Z 809.17,A -85,B 0,C 180,E1 -13710.35,E2 -13710.35} C_VEL
LIN {X 0,Y 347.734,Z 809.172,A -85,B 0,C 180,E1 -13714.045,E2 -13714.045} C_VEL
LIN {X 0,Y 347.741,Z 809.169,A -85,B 0,C 180,E1 -13717.324,E2 -13717.324} C_VEL
LIN {X 0,Y 347.684,Z 809.177,A -85,B 0,C 180,E1 -13720.304,E2 -13720.304} C_VEL
LIN {X 0,Y 347.745,Z 809.192,A -85,B 0,C 180,E1 -13722.81,E2 -13722.81} C_VEL
LIN {X 0,Y 349.493,Z 817.571,A -85,B 0,C 180,E1 -13726.38,E2 -13726.38} C_VEL
LIN {X 0,Y 351.05,Z 825.519,A -85,B 0,C 180,E1 -13729.531,E2 -13729.531} C_VEL
LIN {X 0,Y 352.1,Z 831.485,A -85,B 0,C 180,E1 -13731.777,E2 -13731.777} C_VEL
LIN {X 0,Y 352.157,Z 834.842,A -85,B 0,C 180,E1 -13732.966,E2 -13732.966} C_VEL
LIN {X 0,Y 350.932,Z 845.575,A -85,B 0,C 180,E1 -13736.586,E2 -13736.586} C_VEL
LIN {X 0,Y 349.662,Z 857.468,A -85,B 0,C 180,E1 -13740.502,E2 -13740.502} C_VEL
LIN {X 0,Y 348.663,Z 869.148,A -85,B 0,C 180,E1 -13744.321,E2 -13744.321} C_VEL
LIN {X 0,Y 347.769,Z 882.418,A -85,B 0,C 180,E1 -13748.671,E2 -13748.671} C_VEL
LIN {X 0,Y 347.691,Z 883.515,A -85,B 0,C 180,E1 -13749.035,E2 -13749.035} C_VEL
LIN {X 0,Y 349.617,Z 898.428,A -85,B 0,C 180,E1 -13749.656,E2 -13749.656} C_VEL
LIN {X 0,Y 350.677,Z 910.977,A -85,B 0,C 180,E1 -13750.38,E2 -13750.38} C_VEL
LIN {X 0,Y 351.088,Z 923.621,A -85,B 0,C 180,E1 -13751.322,E2 -13751.322} C_VEL
LIN {X 0,Y 351.448,Z 934.977,A -85,B 0,C 180,E1 -13752.397,E2 -13752.397} C_VEL
LIN {X 0,Y 350.103,Z 946.359,A -85,B 0,C 180,E1 -13753.68,E2 -13753.68} C_VEL
LIN {X 0,Y 349.006,Z 956.633,A -85,B 0,C 180,E1 -13755.147,E2 -13755.147} C_VEL
LIN {X 0,Y 348.238,Z 964.859,A -85,B 0,C 180,E1 -13756.582,E2 -13756.582} C_VEL
LIN {X 0,Y 347.46,Z 973.083,A -85,B 0,C 180,E1 -13758.333,E2 -13758.333} C_VEL
LIN {X 0,Y 347.053,Z 979.729,A -85,B 0,C 180,E1 -13760.091,E2 -13760.091} C_VEL
LIN {X 0,Y 346.88,Z 985.035,A -85,B 0,C 180,E1 -13761.849,E2 -13761.849} C_VEL
LIN {X 0,Y 346.935,Z 988.829,A -85,B 0,C 180,E1 -13763.432,E2 -13763.432} C_VEL
LIN {X 0,Y 347.058,Z 992.277,A -85,B 0,C 180,E1 -13765.356,E2 -13765.356} C_VEL
LIN {X 0,Y 347.132,Z 993.747,A -85,B 0,C 180,E1 -13766.52,E2 -13766.52} C_VEL
LIN {X 0,Y 347.174,Z 994.793,A -85,B 0,C 180,E1 -13767.682,E2 -13767.682} C_VEL
LIN {X 0,Y 347.238,Z 995.436,A -85,B 0,C 180,E1 -13768.842,E2 -13768.842} C_VEL
LIN {X 0,Y 347.29,Z 995.666,A -85,B 0,C 180,E1 -13770.002,E2 -13770.002} C_VEL
LIN {X 0,Y 347.238,Z 995.43,A -85,B 0,C 180,E1 -13771.162,E2 -13771.162} C_VEL
LIN {X 0,Y 347.175,Z 994.783,A -85,B 0,C 180,E1 -13772.322,E2 -13772.322} C_VEL
LIN {X 0,Y 347.133,Z 993.732,A -85,B 0,C 180,E1 -13773.484,E2 -13773.484} C_VEL
LIN {X 0,Y 347.058,Z 992.256,A -85,B 0,C 180,E1 -13774.648,E2 -13774.648} C_VEL
LIN {X 0,Y 346.913,Z 987.985,A -85,B 0,C 180,E1 -13776.937,E2 -13776.937} C_VEL
LIN {X 0,Y 346.932,Z 983.347,A -85,B 0,C 180,E1 -13778.741,E2 -13778.741} C_VEL
LIN {X 0,Y 347.186,Z 977.609,A -85,B 0,C 180,E1 -13780.499,E2 -13780.499} C_VEL
LIN {X 0,Y 347.706,Z 970.493,A -85,B 0,C 180,E1 -13782.255,E2 -13782.255} C_VEL
LIN {X 0,Y 348.486,Z 963.281,A -85,B 0,C 180,E1 -13783.709,E2 -13783.709} C_VEL
LIN {X 0,Y 349.28,Z 954.585,A -85,B 0,C 180,E1 -13785.166,E2 -13785.166} C_VEL
LIN {X 0,Y 350.429,Z 943.911,A -85,B 0,C 180,E1 -13786.608,E2 -13786.608} C_VEL
LIN {X 0,Y 351.468,Z 934.838,A -85,B 0,C 180,E1 -13787.606,E2 -13787.606} C_VEL
LIN {X 0,Y 351.404,Z 921.006,A -85,B 0,C 180,E1 -13789.104,E2 -13789.104} C_VEL
LIN {X 0,Y 351.304,Z 906.986,A -85,B 0,C 180,E1 -13790.342,E2 -13790.342} C_VEL
LIN {X 0,Y 350.854,Z 897.845,A -85,B 0,C 180,E1 -13791.059,E2 -13791.059} C_VEL
LIN {X 0,Y 348.803,Z 883.999,A -85,B 0,C 180,E1 -13792.074,E2 -13792.074} C_VEL
LIN {X 0,Y 347.945,Z 879.027,A -85,B 0,C 180,E1 -13792.438,E2 -13792.438} C_VEL
LIN {X 0,Y 348.8,Z 867.176,A -85,B 0,C 180,E1 -13796.315,E2 -13796.315} C_VEL
LIN {X 0,Y 349.838,Z 855.421,A -85,B 0,C 180,E1 -13800.15,E2 -13800.15} C_VEL
LIN {X 0,Y 351.113,Z 843.513,A -85,B 0,C 180,E1 -13804.089,E2 -13804.089} C_VEL
LIN {X 0,Y 352.148,Z 834.802,A -85,B 0,C 180,E1 -13807.032,E2 -13807.032} C_VEL
LIN {X 0,Y 352.06,Z 831.413,A -85,B 0,C 180,E1 -13808.233,E2 -13808.233} C_VEL
LIN {X 0,Y 350.564,Z 822.998,A -85,B 0,C 180,E1 -13811.422,E2 -13811.422} C_VEL
LIN {X 0,Y 348.847,Z 814.578,A -85,B 0,C 180,E1 -13814.842,E2 -13814.842} C_VEL
LIN {X 0,Y 347.711,Z 809.176,A -85,B 0,C 180,E1 -13817.192,E2 -13817.192} C_VEL
LIN {X 0,Y 347.736,Z 809.167,A -85,B 0,C 180,E1 -13821.205,E2 -13821.205} C_VEL
LIN {X 0,Y 347.787,Z 809.163,A -85,B 0,C 180,E1 -13824.124,E2 -13824.124} C_VEL
LIN {X 0,Y 347.744,Z 809.168,A -85,B 0,C 180,E1 -13828.087,E2 -13828.087} C_VEL
LIN {X 0,Y 347.739,Z 809.171,A -85,B 0,C 180,E1 -13830.984,E2 -13830.984} C_VEL
LIN {X 0,Y 347.736,Z 809.168,A -85,B 0,C 180,E1 -13833.6,E2 -13833.6} C_VEL
LIN {X 0,Y 347.75,Z 809.167,A -85,B 0,C 180,E1 -13836.159,E2 -13836.159} C_VEL
LIN {X 0,Y 347.762,Z 809.196,A -85,B 0,C 180,E1 -13837.571,E2 -13837.571} C_VEL
LIN {X 0,Y 348.891,Z 812.182,A -85,B 0,C 180,E1 -13837.917,E2 -13837.917} C_VEL
LIN {X 0,Y 352.672,Z 819.613,A -85,B 0,C 180,E1 -13838.98,E2 -13838.98} C_VEL
LIN {X 0,Y 356.542,Z 829.933,A -85,B 0,C 180,E1 -13840.422,E2 -13840.422} C_VEL
LIN {X 0,Y 358.22,Z 835.584,A -85,B 0,C 180,E1 -13841.225,E2 -13841.225} C_VEL
LIN {X 0,Y 357.011,Z 846.684,A -85,B 0,C 180,E1 -13842.53,E2 -13842.53} C_VEL
LIN {X 0,Y 355.905,Z 854.684,A -85,B 0,C 180,E1 -13843.657,E2 -13843.657} C_VEL
LIN {X 0,Y 354.625,Z 863.087,A -85,B 0,C 180,E1 -13845.07,E2 -13845.07} C_VEL
LIN {X 0,Y 353.458,Z 869.931,A -85,B 0,C 180,E1 -13846.489,E2 -13846.489} C_VEL
LIN {X 0,Y 352.575,Z 875.174,A -85,B 0,C 180,E1 -13847.772,E2 -13847.772} C_VEL
LIN {X 0,Y 351.753,Z 879.65,A -85,B 0,C 180,E1 -13849.058,E2 -13849.058} C_VEL
LIN {X 0,Y 350.702,Z 884.469,A -85,B 0,C 180,E1 -13850.775,E2 -13850.775} C_VEL
LIN {X 0,Y 349.863,Z 888.087,A -85,B 0,C 180,E1 -13852.497,E2 -13852.497} C_VEL
LIN {X 0,Y 349.233,Z 890.695,A -85,B 0,C 180,E1 -13854.225,E2 -13854.225} C_VEL
LIN {X 0,Y 348.919,Z 891.941,A -85,B 0,C 180,E1 -13855.379,E2 -13855.379} C_VEL
LIN {X 0,Y 348.416,Z 893.085,A -85,B 0,C 180,E1 -13857.688,E2 -13857.688} C_VEL
LIN {X 0,Y 348.139,Z 893.07,A -85,B 0,C 180,E1 -13858.843,E2 -13858.843} C_VEL
LIN {X 0,Y 347.969,Z 892.639,A -85,B 0,C 180,E1 -13860,E2 -13860} C_VEL
LIN {X 0,Y 347.951,Z 891.717,A -85,B 0,C 180,E1 -13861.157,E2 -13861.157} C_VEL
LIN {X 0,Y 347.855,Z 890.449,A -85,B 0,C 180,E1 -13862.316,E2 -13862.316} C_VEL
LIN {X 0,Y 347.887,Z 886.583,A -85,B 0,C 180,E1 -13864.635,E2 -13864.635} C_VEL
LIN {X 0,Y 348.355,Z 882.436,A -85,B 0,C 180,E1 -13866.371,E2 -13866.371} C_VEL
LIN {X 0,Y 348.656,Z 877.156,A -85,B 0,C 180,E1 -13868.112,E2 -13868.112} C_VEL
LIN {X 0,Y 349,Z 871.796,A -85,B 0,C 180,E1 -13869.563,E2 -13869.563} C_VEL
LIN {X 0,Y 349.607,Z 864.029,A -85,B 0,C 180,E1 -13871.303,E2 -13871.303} C_VEL
LIN {X 0,Y 350.14,Z 855.979,A -85,B 0,C 180,E1 -13872.756,E2 -13872.756} C_VEL
LIN {X 0,Y 350.69,Z 848.482,A -85,B 0,C 180,E1 -13873.915,E2 -13873.915} C_VEL
LIN {X 0,Y 351.216,Z 840.881,A -85,B 0,C 180,E1 -13874.93,E2 -13874.93} C_VEL
LIN {X 0,Y 351.946,Z 830.721,A -85,B 0,C 180,E1 -13876.085,E2 -13876.085} C_VEL
LIN {X 0,Y 352.036,Z 825.431,A -85,B 0,C 180,E1 -13876.607,E2 -13876.607} C_VEL
LIN {X 0,Y 348.849,Z 813.234,A -85,B 0,C 180,E1 -13877.749,E2 -13877.749} C_VEL
LIN {X 0,Y 347.792,Z 809.161,A -85,B 0,C 180,E1 -13878.098,E2 -13878.098} C_VEL
LIN {X 0,Y 347.753,Z 809.159,A -85,B 0,C 180,E1 -13881.617,E2 -13881.617} C_VEL
LIN {X 0,Y 347.74,Z 809.166,A -85,B 0,C 180,E1 -13885.114,E2 -13885.114} C_VEL
LIN {X 0,Y 347.731,Z 809.162,A -85,B 0,C 180,E1 -13887.701,E2 -13887.701} C_VEL
LIN {X 0,Y 347.745,Z 809.164,A -85,B 0,C 180,E1 -13890.348,E2 -13890.348} C_VEL
LIN {X 0,Y 347.755,Z 809.164,A -85,B 0,C 180,E1 -13894.043,E2 -13894.043} C_VEL
LIN {X 0,Y 347.761,Z 809.16,A -85,B 0,C 180,E1 -13897.321,E2 -13897.321} C_VEL
LIN {X 0,Y 347.748,Z 809.166,A -85,B 0,C 180,E1 -13901.6,E2 -13901.6} C_VEL
LIN {X 0,Y 347.712,Z 809.169,A -85,B 0,C 180,E1 -13905.026,E2 -13905.026} C_VEL
LIN {X 0,Y 347.748,Z 809.168,A -85,B 0,C 180,E1 -13908.398,E2 -13908.398} C_VEL
LIN {X 0,Y 347.763,Z 809.162,A -85,B 0,C 180,E1 -13912.677,E2 -13912.677} C_VEL
LIN {X 0,Y 347.755,Z 809.167,A -85,B 0,C 180,E1 -13915.955,E2 -13915.955} C_VEL
LIN {X 0,Y 347.756,Z 809.161,A -85,B 0,C 180,E1 -13919.651,E2 -13919.651} C_VEL
LIN {X 0,Y 347.837,Z 809.15,A -85,B 0,C 180,E1 -13923.606,E2 -13923.606} C_VEL
LIN {X 0,Y 347.795,Z 809.152,A -85,B 0,C 180,E1 -13926.16,E2 -13926.16} C_VEL
LIN {X 0,Y 347.814,Z 809.164,A -85,B 0,C 180,E1 -13929.937,E2 -13929.937} C_VEL
LIN {X 0,Y 352.243,Z 822.145,A -85,B 0,C 180,E1 -13931.139,E2 -13931.139} C_VEL
LIN {X 0,Y 354.942,Z 831.278,A -85,B 0,C 180,E1 -13932.136,E2 -13932.136} C_VEL
LIN {X 0,Y 355.023,Z 833.815,A -85,B 0,C 180,E1 -13932.396,E2 -13932.396} C_VEL
LIN {X 0,Y 353.986,Z 844.403,A -85,B 0,C 180,E1 -13933.564,E2 -13933.564} C_VEL
LIN {X 0,Y 352.966,Z 854.741,A -85,B 0,C 180,E1 -13934.997,E2 -13934.997} C_VEL
LIN {X 0,Y 352.011,Z 863.107,A -85,B 0,C 180,E1 -13936.431,E2 -13936.431} C_VEL
LIN {X 0,Y 350.943,Z 871.225,A -85,B 0,C 180,E1 -13938.153,E2 -13938.153} C_VEL
LIN {X 0,Y 350.114,Z 877.875,A -85,B 0,C 180,E1 -13939.923,E2 -13939.923} C_VEL
LIN {X 0,Y 349.4,Z 883.697,A -85,B 0,C 180,E1 -13941.904,E2 -13941.904} C_VEL
LIN {X 0,Y 348.678,Z 887.591,A -85,B 0,C 180,E1 -13943.633,E2 -13943.633} C_VEL
LIN {X 0,Y 348.276,Z 890.443,A -85,B 0,C 180,E1 -13945.368,E2 -13945.368} C_VEL
LIN {X 0,Y 348.271,Z 891.785,A -85,B 0,C 180,E1 -13946.527,E2 -13946.527} C_VEL
LIN {X 0,Y 348.038,Z 893.359,A -85,B 0,C 180,E1 -13948.841,E2 -13948.841} C_VEL
LIN {X 0,Y 347.997,Z 893.59,A -85,B 0,C 180,E1 -13949.998,E2 -13949.998} C_VEL
LIN {X 0,Y 348.147,Z 892.829,A -85,B 0,C 180,E1 -13952.312,E2 -13952.312} C_VEL
LIN {X 0,Y 348.264,Z 890.593,A -85,B 0,C 180,E1 -13954.628,E2 -13954.628} C_VEL
LIN {X 0,Y 348.667,Z 887.788,A -85,B 0,C 180,E1 -13956.363,E2 -13956.363} C_VEL
LIN {X 0,Y 349.419,Z 883.95,A -85,B 0,C 180,E1 -13958.092,E2 -13958.092} C_VEL
LIN {X 0,Y 350.153,Z 878.23,A -85,B 0,C 180,E1 -13960.072,E2 -13960.072} C_VEL
LIN {X 0,Y 350.886,Z 871.673,A -85,B 0,C 180,E1 -13961.845,E2 -13961.845} C_VEL
LIN {X 0,Y 351.953,Z 863.649,A -85,B 0,C 180,E1 -13963.568,E2 -13963.568} C_VEL
LIN {X 0,Y 352.873,Z 855.431,A -85,B 0,C 180,E1 -13965.003,E2 -13965.003} C_VEL
LIN {X 0,Y 353.928,Z 845.25,A -85,B 0,C 180,E1 -13966.435,E2 -13966.435} C_VEL
LIN {X 0,Y 354.977,Z 834.779,A -85,B 0,C 180,E1 -13967.609,E2 -13967.609} C_VEL
LIN {X 0,Y 355.068,Z 831.922,A -85,B 0,C 180,E1 -13967.899,E2 -13967.899} C_VEL
LIN {X 0,Y 351.867,Z 820.992,A -85,B 0,C 180,E1 -13969.082,E2 -13969.082} C_VEL
LIN {X 0,Y 347.85,Z 809.156,A -85,B 0,C 180,E1 -13970.163,E2 -13970.163} C_VEL
LIN {X 0,Y 347.813,Z 809.159,A -85,B 0,C 180,E1 -13974.593,E2 -13974.593} C_VEL
LIN {X 0,Y 347.806,Z 809.163,A -85,B 0,C 180,E1 -13977.691,E2 -13977.691} C_VEL
LIN {X 0,Y 347.758,Z 809.168,A -85,B 0,C 180,E1 -13980.344,E2 -13980.344} C_VEL
LIN {X 0,Y 347.737,Z 809.171,A -85,B 0,C 180,E1 -13984.462,E2 -13984.462} C_VEL
LIN {X 0,Y 347.768,Z 809.168,A -85,B 0,C 180,E1 -13987.987,E2 -13987.987} C_VEL
LIN {X 0,Y 347.777,Z 809.164,A -85,B 0,C 180,E1 -13991.823,E2 -13991.823} C_VEL
LIN {X 0,Y 347.761,Z 809.162,A -85,B 0,C 180,E1 -13992.273,E2 -13992.273} C_VEL
LIN {X 0,Y 347.099,Z 809.247,A -85,B 0,C 180,E1 -13993.241,E2 -13993.241} C_VEL
LIN {X 0,Y 344.267,Z 809.602,A -85,B 0,C 180,E1 -13994.815,E2 -13994.815} C_VEL
LIN {X 0,Y 341.864,Z 809.902,A -85,B 0,C 180,E1 -13996.089,E2 -13996.089} C_VEL
LIN {X 0,Y 340.826,Z 810.024,A -85,B 0,C 180,E1 -13997.075,E2 -13997.075} C_VEL
LIN {X 0,Y 340.739,Z 810.034,A -85,B 0,C 180,E1 -13997.409,E2 -13997.409} C_VEL
LIN {X 0,Y 340.725,Z 810.044,A -85,B 0,C 180,E1 -14000.251,E2 -14000.251} C_VEL
LIN {X 0,Y 340.701,Z 810.043,A -85,B 0,C 180,E1 -14003.557,E2 -14003.557} C_VEL
LIN {X 0,Y 340.679,Z 810.042,A -85,B 0,C 180,E1 -14006.152,E2 -14006.152} C_VEL
LIN {X 0,Y 340.761,Z 810.032,A -85,B 0,C 180,E1 -14010.331,E2 -14010.331} C_VEL
LIN {X 0,Y 340.791,Z 810.033,A -85,B 0,C 180,E1 -14013.019,E2 -14013.019} C_VEL
LIN {X 0,Y 340.714,Z 810.047,A -85,B 0,C 180,E1 -14016.926,E2 -14016.926} C_VEL
LIN {X 0,Y 340.775,Z 810.034,A -85,B 0,C 180,E1 -14020.732,E2 -14020.732} C_VEL
LIN {X 0,Y 340.771,Z 810.033,A -85,B 0,C 180,E1 -14023.218,E2 -14023.218} C_VEL
LIN {X 0,Y 340.831,Z 810.028,A -85,B 0,C 180,E1 -14026.89,E2 -14026.89} C_VEL
LIN {X 0,Y 340.911,Z 810.013,A -85,B 0,C 180,E1 -14030.507,E2 -14030.507} C_VEL
LIN {X 0,Y 341.043,Z 810.003,A -85,B 0,C 180,E1 -14032.897,E2 -14032.897} C_VEL
LIN {X 0,Y 341.152,Z 809.989,A -85,B 0,C 180,E1 -14037.639,E2 -14037.639} C_VEL
LIN {X 0,Y 341.279,Z 809.976,A -85,B 0,C 180,E1 -14040,E2 -14040} C_VEL
LIN {X 0,Y 341.151,Z 809.991,A -85,B 0,C 180,E1 -14042.361,E2 -14042.361} C_VEL
LIN {X 0,Y 341.033,Z 810.003,A -85,B 0,C 180,E1 -14047.103,E2 -14047.103} C_VEL
LIN {X 0,Y 340.858,Z 810.023,A -85,B 0,C 180,E1 -14050.694,E2 -14050.694} C_VEL
LIN {X 0,Y 340.847,Z 810.028,A -85,B 0,C 180,E1 -14054.326,E2 -14054.326} C_VEL
LIN {X 0,Y 340.821,Z 810.032,A -85,B 0,C 180,E1 -14058.467,E2 -14058.467} C_VEL
LIN {X 0,Y 340.702,Z 810.048,A -85,B 0,C 180,E1 -14061.843,E2 -14061.843} C_VEL
LIN {X 0,Y 340.703,Z 810.045,A -85,B 0,C 180,E1 -14065.67,E2 -14065.67} C_VEL
LIN {X 0,Y 340.69,Z 810.048,A -85,B 0,C 180,E1 -14069.676,E2 -14069.676} C_VEL
LIN {X 0,Y 340.672,Z 810.048,A -85,B 0,C 180,E1 -14072.437,E2 -14072.437} C_VEL
LIN {X 0,Y 340.701,Z 810.045,A -85,B 0,C 180,E1 -14075.281,E2 -14075.281} C_VEL
LIN {X 0,Y 340.679,Z 810.049,A -85,B 0,C 180,E1 -14078.384,E2 -14078.384} C_VEL
LIN {X 0,Y 340.712,Z 810.16,A -85,B 0,C 180,E1 -14082.361,E2 -14082.361} C_VEL
LIN {X 0,Y 342.409,Z 818.289,A -85,B 0,C 180,E1 -14085.921,E2 -14085.921} C_VEL
LIN {X 0,Y 343.982,Z 826.269,A -85,B 0,C 180,E1 -14089.175,E2 -14089.175} C_VEL
LIN {X 0,Y 345.22,Z 833.591,A -85,B 0,C 180,E1 -14091.991,E2 -14091.991} C_VEL
LIN {X 0,Y 345.081,Z 836.878,A -85,B 0,C 180,E1 -14093.166,E2 -14093.166} C_VEL
LIN {X 0,Y 343.739,Z 847.911,A -85,B 0,C 180,E1 -14096.959,E2 -14096.959} C_VEL
LIN {X 0,Y 342.397,Z 860.368,A -85,B 0,C 180,E1 -14101.163,E2 -14101.163} C_VEL
LIN {X 0,Y 341.467,Z 871.534,A -85,B 0,C 180,E1 -14104.904,E2 -14104.904} C_VEL
LIN {X 0,Y 340.69,Z 882.436,A -85,B 0,C 180,E1 -14108.583,E2 -14108.583} C_VEL
LIN {X 0,Y 342.661,Z 897.348,A -85,B 0,C 180,E1 -14109.224,E2 -14109.224} C_VEL
LIN {X 0,Y 343.741,Z 909.904,A -85,B 0,C 180,E1 -14109.968,E2 -14109.968} C_VEL
LIN {X 0,Y 344.17,Z 922.553,A -85,B 0,C 180,E1 -14110.933,E2 -14110.933} C_VEL
LIN {X 0,Y 344.494,Z 933.909,A -85,B 0,C 180,E1 -14112.03,E2 -14112.03} C_VEL
LIN {X 0,Y 343.749,Z 941.789,A -85,B 0,C 180,E1 -14112.911,E2 -14112.911} C_VEL
LIN {X 0,Y 342.584,Z 951.64,A -85,B 0,C 180,E1 -14114.23,E2 -14114.23} C_VEL
LIN {X 0,Y 341.596,Z 958.867,A -85,B 0,C 180,E1 -14115.387,E2 -14115.387} C_VEL
LIN {X 0,Y 341.31,Z 963.814,A -85,B 0,C 180,E1 -14116.305,E2 -14116.305} C_VEL
LIN {X 0,Y 340.475,Z 972.037,A -85,B 0,C 180,E1 -14118.09,E2 -14118.09} C_VEL
LIN {X 0,Y 340.021,Z 978.681,A -85,B 0,C 180,E1 -14119.884,E2 -14119.884} C_VEL
LIN {X 0,Y 339.812,Z 983.988,A -85,B 0,C 180,E1 -14121.678,E2 -14121.678} C_VEL
LIN {X 0,Y 339.888,Z 987.993,A -85,B 0,C 180,E1 -14123.392,E2 -14123.392} C_VEL
LIN {X 0,Y 340,Z 991.237,A -85,B 0,C 180,E1 -14125.259,E2 -14125.259} C_VEL
LIN {X 0,Y 340.089,Z 992.711,A -85,B 0,C 180,E1 -14126.448,E2 -14126.448} C_VEL
LIN {X 0,Y 340.135,Z 993.759,A -85,B 0,C 180,E1 -14127.634,E2 -14127.634} C_VEL
LIN {X 0,Y 340.206,Z 994.403,A -85,B 0,C 180,E1 -14128.818,E2 -14128.818} C_VEL
LIN {X 0,Y 340.265,Z 994.635,A -85,B 0,C 180,E1 -14130.002,E2 -14130.002} C_VEL
LIN {X 0,Y 340.206,Z 994.397,A -85,B 0,C 180,E1 -14131.186,E2 -14131.186} C_VEL
LIN {X 0,Y 340.136,Z 993.748,A -85,B 0,C 180,E1 -14132.37,E2 -14132.37} C_VEL
LIN {X 0,Y 340.09,Z 992.696,A -85,B 0,C 180,E1 -14133.556,E2 -14133.556} C_VEL
LIN {X 0,Y 340.001,Z 991.216,A -85,B 0,C 180,E1 -14134.745,E2 -14134.745} C_VEL
LIN {X 0,Y 339.846,Z 987.215,A -85,B 0,C 180,E1 -14136.956,E2 -14136.956} C_VEL
LIN {X 0,Y 339.869,Z 982.297,A -85,B 0,C 180,E1 -14138.924,E2 -14138.924} C_VEL
LIN {X 0,Y 340.13,Z 976.554,A -85,B 0,C 180,E1 -14140.719,E2 -14140.719} C_VEL
LIN {X 0,Y 340.702,Z 969.439,A -85,B 0,C 180,E1 -14142.511,E2 -14142.511} C_VEL
LIN {X 0,Y 341.646,Z 960.588,A -85,B 0,C 180,E1 -14144.293,E2 -14144.293} C_VEL
LIN {X 0,Y 342.698,Z 950.554,A -85,B 0,C 180,E1 -14145.922,E2 -14145.922} C_VEL
LIN {X 0,Y 344.251,Z 938.274,A -85,B 0,C 180,E1 -14147.527,E2 -14147.527} C_VEL
LIN {X 0,Y 344.517,Z 933.427,A -85,B 0,C 180,E1 -14148.127,E2 -14148.127} C_VEL
LIN {X 0,Y 344.613,Z 924.591,A -85,B 0,C 180,E1 -14149.16,E2 -14149.16} C_VEL
LIN {X 0,Y 344.807,Z 915.179,A -85,B 0,C 180,E1 -14150.117,E2 -14150.117} C_VEL
LIN {X 0,Y 344.822,Z 904.604,A -85,B 0,C 180,E1 -14151.054,E2 -14151.054} C_VEL
LIN {X 0,Y 343.878,Z 894.108,A -85,B 0,C 180,E1 -14151.931,E2 -14151.931} C_VEL
LIN {X 0,Y 341.721,Z 881.243,A -85,B 0,C 180,E1 -14152.947,E2 -14152.947} C_VEL
LIN {X 0,Y 340.996,Z 876.864,A -85,B 0,C 180,E1 -14153.296,E2 -14153.296} C_VEL
LIN {X 0,Y 341.872,Z 866.152,A -85,B 0,C 180,E1 -14156.891,E2 -14156.891} C_VEL
LIN {X 0,Y 342.97,Z 854.434,A -85,B 0,C 180,E1 -14160.818,E2 -14160.818} C_VEL
LIN {X 0,Y 344.1,Z 844.545,A -85,B 0,C 180,E1 -14164.173,E2 -14164.173} C_VEL
LIN {X 0,Y 345.232,Z 835.094,A -85,B 0,C 180,E1 -14167.445,E2 -14167.445} C_VEL
LIN {X 0,Y 344.721,Z 830.338,A -85,B 0,C 180,E1 -14169.22,E2 -14169.22} C_VEL
LIN {X 0,Y 343.123,Z 821.972,A -85,B 0,C 180,E1 -14172.528,E2 -14172.528} C_VEL
LIN {X 0,Y 341.236,Z 812.701,A -85,B 0,C 180,E1 -14176.473,E2 -14176.473} C_VEL
LIN {X 0,Y 340.67,Z 810.051,A -85,B 0,C 180,E1 -14177.703,E2 -14177.703} C_VEL
LIN {X 0,Y 340.723,Z 810.041,A -85,B 0,C 180,E1 -14181.771,E2 -14181.771} C_VEL
LIN {X 0,Y 340.727,Z 810.04,A -85,B 0,C 180,E1 -14185.597,E2 -14185.597} C_VEL
LIN {X 0,Y 340.697,Z 810.048,A -85,B 0,C 180,E1 -14188.955,E2 -14188.955} C_VEL
LIN {X 0,Y 340.714,Z 810.046,A -85,B 0,C 180,E1 -14193.012,E2 -14193.012} C_VEL
LIN {X 0,Y 340.694,Z 810.134,A -85,B 0,C 180,E1 -14196.643,E2 -14196.643} C_VEL
LIN {X 0,Y 341.804,Z 813.069,A -85,B 0,C 180,E1 -14197.004,E2 -14197.004} C_VEL
LIN {X 0,Y 342.88,Z 814.576,A -85,B 0,C 180,E1 -14197.277,E2 -14197.277} C_VEL
LIN {X 0,Y 347.148,Z 823.568,A -85,B 0,C 180,E1 -14198.637,E2 -14198.637} C_VEL
LIN {X 0,Y 350.224,Z 831.893,A -85,B 0,C 180,E1 -14199.874,E2 -14199.874} C_VEL
LIN {X 0,Y 352.033,Z 838.736,A -85,B 0,C 180,E1 -14200.882,E2 -14200.882} C_VEL
LIN {X 0,Y 350.62,Z 849.393,A -85,B 0,C 180,E1 -14202.201,E2 -14202.201} C_VEL
LIN {X 0,Y 349.436,Z 857.141,A -85,B 0,C 180,E1 -14203.345,E2 -14203.345} C_VEL
LIN {X 0,Y 348.088,Z 865.355,A -85,B 0,C 180,E1 -14204.783,E2 -14204.783} C_VEL
LIN {X 0,Y 346.833,Z 872.1,A -85,B 0,C 180,E1 -14206.256,E2 -14206.256} C_VEL
LIN {X 0,Y 345.747,Z 877.865,A -85,B 0,C 180,E1 -14207.76,E2 -14207.76} C_VEL
LIN {X 0,Y 344.594,Z 883.075,A -85,B 0,C 180,E1 -14209.423,E2 -14209.423} C_VEL
LIN {X 0,Y 343.646,Z 887.42,A -85,B 0,C 180,E1 -14211.177,E2 -14211.177} C_VEL
LIN {X 0,Y 342.616,Z 890.579,A -85,B 0,C 180,E1 -14212.93,E2 -14212.93} C_VEL
LIN {X 0,Y 341.988,Z 893.312,A -85,B 0,C 180,E1 -14215.285,E2 -14215.285} C_VEL
LIN {X 0,Y 341.441,Z 894.307,A -85,B 0,C 180,E1 -14217.641,E2 -14217.641} C_VEL
LIN {X 0,Y 341.166,Z 894.233,A -85,B 0,C 180,E1 -14218.82,E2 -14218.82} C_VEL
LIN {X 0,Y 340.952,Z 893.715,A -85,B 0,C 180,E1 -14220,E2 -14220} C_VEL
LIN {X 0,Y 340.831,Z 891.429,A -85,B 0,C 180,E1 -14222.364,E2 -14222.364} C_VEL
LIN {X 0,Y 340.798,Z 888.605,A -85,B 0,C 180,E1 -14224.139,E2 -14224.139} C_VEL
LIN {X 0,Y 341.188,Z 884.726,A -85,B 0,C 180,E1 -14225.912,E2 -14225.912} C_VEL
LIN {X 0,Y 341.602,Z 878.728,A -85,B 0,C 180,E1 -14227.983,E2 -14227.983} C_VEL
LIN {X 0,Y 342.014,Z 872.222,A -85,B 0,C 180,E1 -14229.76,E2 -14229.76} C_VEL
LIN {X 0,Y 342.535,Z 865.75,A -85,B 0,C 180,E1 -14231.24,E2 -14231.24} C_VEL
LIN {X 0,Y 343.099,Z 857.842,A -85,B 0,C 180,E1 -14232.721,E2 -14232.721} C_VEL
LIN {X 0,Y 343.701,Z 849.465,A -85,B 0,C 180,E1 -14234.053,E2 -14234.053} C_VEL
LIN {X 0,Y 344.238,Z 841.853,A -85,B 0,C 180,E1 -14235.088,E2 -14235.088} C_VEL
LIN {X 0,Y 344.993,Z 831.687,A -85,B 0,C 180,E1 -14236.267,E2 -14236.267} C_VEL
LIN {X 0,Y 345.029,Z 826.538,A -85,B 0,C 180,E1 -14236.788,E2 -14236.788} C_VEL
LIN {X 0,Y 341.822,Z 814.253,A -85,B 0,C 180,E1 -14237.963,E2 -14237.963} C_VEL
LIN {X 0,Y 340.748,Z 810.037,A -85,B 0,C 180,E1 -14238.324,E2 -14238.324} C_VEL
LIN {X 0,Y 340.726,Z 810.035,A -85,B 0,C 180,E1 -14241.841,E2 -14241.841} C_VEL
LIN {X 0,Y 340.711,Z 810.041,A -85,B 0,C 180,E1 -14244.82,E2 -14244.82} C_VEL
LIN {X 0,Y 340.682,Z 810.043,A -85,B 0,C 180,E1 -14248.325,E2 -14248.325} C_VEL
LIN {X 0,Y 340.7,Z 810.041,A -85,B 0,C 180,E1 -14251.045,E2 -14251.045} C_VEL
LIN {X 0,Y 340.722,Z 810.039,A -85,B 0,C 180,E1 -14255.279,E2 -14255.279} C_VEL
LIN {X 0,Y 340.7,Z 810.042,A -85,B 0,C 180,E1 -14258.382,E2 -14258.382} C_VEL
LIN {X 0,Y 340.7,Z 810.041,A -85,B 0,C 180,E1 -14262.043,E2 -14262.043} C_VEL
LIN {X 0,Y 340.658,Z 810.048,A -85,B 0,C 180,E1 -14266.226,E2 -14266.226} C_VEL
LIN {X 0,Y 340.678,Z 810.047,A -85,B 0,C 180,E1 -14268.687,E2 -14268.687} C_VEL
LIN {X 0,Y 340.725,Z 810.043,A -85,B 0,C 180,E1 -14271.77,E2 -14271.77} C_VEL
LIN {X 0,Y 340.73,Z 810.04,A -85,B 0,C 180,E1 -14275.594,E2 -14275.594} C_VEL
LIN {X 0,Y 340.705,Z 810.04,A -85,B 0,C 180,E1 -14278.954,E2 -14278.954} C_VEL
LIN {X 0,Y 340.81,Z 810.025,A -85,B 0,C 180,E1 -14283.019,E2 -14283.019} C_VEL
LIN {X 0,Y 340.736,Z 810.04,A -85,B 0,C 180,E1 -14286.926,E2 -14286.926} C_VEL
LIN {X 0,Y 340.793,Z 810.145,A -85,B 0,C 180,E1 -14289.508,E2 -14289.508} C_VEL
LIN {X 0,Y 344.244,Z 819.999,A -85,B 0,C 180,E1 -14290.412,E2 -14290.412} C_VEL
LIN {X 0,Y 347.477,Z 830.345,A -85,B 0,C 180,E1 -14291.531,E2 -14291.531} C_VEL
LIN {X 0,Y 348.392,Z 833.895,A -85,B 0,C 180,E1 -14291.947,E2 -14291.947} C_VEL
LIN {X 0,Y 347.384,Z 844.284,A -85,B 0,C 180,E1 -14293.091,E2 -14293.091} C_VEL
LIN {X 0,Y 346.351,Z 853.872,A -85,B 0,C 180,E1 -14294.401,E2 -14294.401} C_VEL
LIN {X 0,Y 345.356,Z 862.57,A -85,B 0,C 180,E1 -14295.864,E2 -14295.864} C_VEL
LIN {X 0,Y 344.383,Z 869.748,A -85,B 0,C 180,E1 -14297.325,E2 -14297.325} C_VEL
LIN {X 0,Y 343.449,Z 877.117,A -85,B 0,C 180,E1 -14299.182,E2 -14299.182} C_VEL
LIN {X 0,Y 342.696,Z 883.169,A -85,B 0,C 180,E1 -14301.15,E2 -14301.15} C_VEL
LIN {X 0,Y 341.837,Z 887.432,A -85,B 0,C 180,E1 -14302.912,E2 -14302.912} C_VEL
LIN {X 0,Y 341.545,Z 889.658,A -85,B 0,C 180,E1 -14304.093,E2 -14304.093} C_VEL
LIN {X 0,Y 341.275,Z 891.475,A -85,B 0,C 180,E1 -14305.273,E2 -14305.273} C_VEL
LIN {X 0,Y 341.273,Z 892.815,A -85,B 0,C 180,E1 -14306.456,E2 -14306.456} C_VEL
LIN {X 0,Y 341.017,Z 894.391,A -85,B 0,C 180,E1 -14308.817,E2 -14308.817} C_VEL
LIN {X 0,Y 340.974,Z 894.621,A -85,B 0,C 180,E1 -14309.998,E2 -14309.998} C_VEL
LIN {X 0,Y 341.133,Z 893.859,A -85,B 0,C 180,E1 -14312.359,E2 -14312.359} C_VEL
LIN {X 0,Y 341.218,Z 892.925,A -85,B 0,C 180,E1 -14313.54,E2 -14313.54} C_VEL
LIN {X 0,Y 341.263,Z 891.624,A -85,B 0,C 180,E1 -14314.723,E2 -14314.723} C_VEL
LIN {X 0,Y 341.686,Z 888.819,A -85,B 0,C 180,E1 -14316.493,E2 -14316.493} C_VEL
LIN {X 0,Y 342.468,Z 884.98,A -85,B 0,C 180,E1 -14318.257,E2 -14318.257} C_VEL
LIN {X 0,Y 343.12,Z 880.556,A -85,B 0,C 180,E1 -14319.859,E2 -14319.859} C_VEL
LIN {X 0,Y 343.841,Z 873.904,A -85,B 0,C 180,E1 -14321.792,E2 -14321.792} C_VEL
LIN {X 0,Y 344.934,Z 866.129,A -85,B 0,C 180,E1 -14323.549,E2 -14323.549} C_VEL
LIN {X 0,Y 345.917,Z 858.2,A -85,B 0,C 180,E1 -14325.011,E2 -14325.011} C_VEL
LIN {X 0,Y 346.982,Z 848.51,A -85,B 0,C 180,E1 -14326.471,E2 -14326.471} C_VEL
LIN {X 0,Y 348.034,Z 837.849,A -85,B 0,C 180,E1 -14327.752,E2 -14327.752} C_VEL
LIN {X 0,Y 348.335,Z 833.485,A -85,B 0,C 180,E1 -14328.205,E2 -14328.205} C_VEL
LIN {X 0,Y 345.16,Z 822.724,A -85,B 0,C 180,E1 -14329.412,E2 -14329.412} C_VEL
LIN {X 0,Y 341.114,Z 811.373,A -85,B 0,C 180,E1 -14330.5,E2 -14330.5} C_VEL
LIN {X 0,Y 340.79,Z 810.033,A -85,B 0,C 180,E1 -14330.639,E2 -14330.639} C_VEL
LIN {X 0,Y 340.763,Z 810.037,A -85,B 0,C 180,E1 -14334.841,E2 -14334.841} C_VEL
LIN {X 0,Y 340.774,Z 810.037,A -85,B 0,C 180,E1 -14337.523,E2 -14337.523} C_VEL
LIN {X 0,Y 340.698,Z 810.045,A -85,B 0,C 180,E1 -14341.042,E2 -14341.042} C_VEL
LIN {X 0,Y 340.711,Z 810.044,A -85,B 0,C 180,E1 -14345.276,E2 -14345.276} C_VEL
LIN {X 0,Y 340.71,Z 810.047,A -85,B 0,C 180,E1 -14348.386,E2 -14348.386} C_VEL
LIN {X 0,Y 340.718,Z 810.041,A -85,B 0,C 180,E1 -14351.301,E2 -14351.301} C_VEL
LIN {X 0,Y 340.772,Z 810.039,A -85,B 0,C 180,E1 -14354.52,E2 -14354.52} C_VEL
LIN {X 0,Y 340.739,Z 810.034,A -85,B 0,C 180,E1 -14357.409,E2 -14357.409} C_VEL
LIN {X 0,Y 340.058,Z 810.125,A -85,B 0,C 180,E1 -14358.396,E2 -14358.396} C_VEL
LIN {X 0,Y 337.186,Z 810.483,A -85,B 0,C 180,E1 -14360.002,E2 -14360.002} C_VEL
LIN {X 0,Y 334.761,Z 810.783,A -85,B 0,C 180,E1 -14361.302,E2 -14361.302} C_VEL
LIN {X 0,Y 333.726,Z 810.911,A -85,B 0,C 180,E1 -14362.309,E2 -14362.309} C_VEL
LIN {X 0,Y 333.644,Z 810.921,A -85,B 0,C 180,E1 -14362.65,E2 -14362.65} C_VEL
LIN {X 0,Y 333.662,Z 810.914,A -85,B 0,C 180,E1 -14365.34,E2 -14365.34} C_VEL
LIN {X 0,Y 333.689,Z 810.912,A -85,B 0,C 180,E1 -14369.709,E2 -14369.709} C_VEL
LIN {X 0,Y 333.73,Z 810.914,A -85,B 0,C 180,E1 -14372.4,E2 -14372.4} C_VEL
LIN {X 0,Y 333.712,Z 810.914,A -85,B 0,C 180,E1 -14375.089,E2 -14375.089} C_VEL
LIN {X 0,Y 333.669,Z 810.918,A -85,B 0,C 180,E1 -14379.018,E2 -14379.018} C_VEL
LIN {X 0,Y 333.778,Z 810.907,A -85,B 0,C 180,E1 -14381.588,E2 -14381.588} C_VEL
LIN {X 0,Y 333.792,Z 810.903,A -85,B 0,C 180,E1 -14385.576,E2 -14385.576} C_VEL
LIN {X 0,Y 333.822,Z 810.904,A -85,B 0,C 180,E1 -14389.078,E2 -14389.078} C_VEL
LIN {X 0,Y 333.996,Z 810.88,A -85,B 0,C 180,E1 -14392.747,E2 -14392.747} C_VEL
LIN {X 0,Y 333.793,Z 810.91,A -85,B 0,C 180,E1 -14395.169,E2 -14395.169} C_VEL
LIN {X 0,Y 334.09,Z 810.868,A -85,B 0,C 180,E1 -14397.589,E2 -14397.589} C_VEL
LIN {X 0,Y 334.23,Z 810.854,A -85,B 0,C 180,E1 -14400,E2 -14400} C_VEL
LIN {X 0,Y 334.088,Z 810.871,A -85,B 0,C 180,E1 -14402.411,E2 -14402.411} C_VEL
LIN {X 0,Y 333.987,Z 810.882,A -85,B 0,C 180,E1 -14407.253,E2 -14407.253} C_VEL
LIN {X 0,Y 333.821,Z 810.9,A -85,B 0,C 180,E1 -14410.922,E2 -14410.922} C_VEL
LIN {X 0,Y 333.792,Z 810.905,A -85,B 0,C 180,E1 -14414.635,E2 -14414.635} C_VEL
LIN {X 0,Y 333.78,Z 810.908,A -85,B 0,C 180,E1 -14418.656,E2 -14418.656} C_VEL
LIN {X 0,Y 333.637,Z 810.928,A -85,B 0,C 180,E1 -14422.282,E2 -14422.282} C_VEL
LIN {X 0,Y 333.672,Z 810.919,A -85,B 0,C 180,E1 -14425.09,E2 -14425.09} C_VEL
LIN {X 0,Y 333.638,Z 810.925,A -85,B 0,C 180,E1 -14428.979,E2 -14428.979} C_VEL
LIN {X 0,Y 333.629,Z 810.925,A -85,B 0,C 180,E1 -14432.588,E2 -14432.588} C_VEL
LIN {X 0,Y 333.659,Z 810.925,A -85,B 0,C 180,E1 -14436.141,E2 -14436.141} C_VEL
LIN {X 0,Y 333.607,Z 810.931,A -85,B 0,C 180,E1 -14439.198,E2 -14439.198} C_VEL
LIN {X 0,Y 333.663,Z 811.055,A -85,B 0,C 180,E1 -14441.87,E2 -14441.87} C_VEL
LIN {X 0,Y 335.322,Z 819.008,A -85,B 0,C 180,E1 -14445.447,E2 -14445.447} C_VEL
LIN {X 0,Y 336.85,Z 826.708,A -85,B 0,C 180,E1 -14448.686,E2 -14448.686} C_VEL
LIN {X 0,Y 338.101,Z 833.597,A -85,B 0,C 180,E1 -14451.424,E2 -14451.424} C_VEL
LIN {X 0,Y 338.273,Z 836.573,A -85,B 0,C 180,E1 -14452.541,E2 -14452.541} C_VEL
LIN {X 0,Y 336.823,Z 847.988,A -85,B 0,C 180,E1 -14456.577,E2 -14456.577} C_VEL
LIN {X 0,Y 335.33,Z 861.285,A -85,B 0,C 180,E1 -14461.184,E2 -14461.184} C_VEL
LIN {X 0,Y 334.422,Z 871.353,A -85,B 0,C 180,E1 -14464.644,E2 -14464.644} C_VEL
LIN {X 0,Y 333.671,Z 881.347,A -85,B 0,C 180,E1 -14468.1,E2 -14468.1} C_VEL
LIN {X 0,Y 335.749,Z 896.728,A -85,B 0,C 180,E1 -14468.796,E2 -14468.796} C_VEL
LIN {X 0,Y 336.879,Z 910.116,A -85,B 0,C 180,E1 -14469.63,E2 -14469.63} C_VEL
LIN {X 0,Y 337.292,Z 921.489,A -85,B 0,C 180,E1 -14470.528,E2 -14470.528} C_VEL
LIN {X 0,Y 337.376,Z 931.346,A -85,B 0,C 180,E1 -14471.48,E2 -14471.48} C_VEL
LIN {X 0,Y 337.419,Z 936.969,A -85,B 0,C 180,E1 -14472.111,E2 -14472.111} C_VEL
LIN {X 0,Y 336.047,Z 947.535,A -85,B 0,C 180,E1 -14473.447,E2 -14473.447} C_VEL
LIN {X 0,Y 334.797,Z 957.46,A -85,B 0,C 180,E1 -14475.014,E2 -14475.014} C_VEL
LIN {X 0,Y 333.937,Z 965.688,A -85,B 0,C 180,E1 -14476.617,E2 -14476.617} C_VEL
LIN {X 0,Y 333.247,Z 973.337,A -85,B 0,C 180,E1 -14478.445,E2 -14478.445} C_VEL
LIN {X 0,Y 332.89,Z 979.522,A -85,B 0,C 180,E1 -14480.279,E2 -14480.279} C_VEL
LIN {X 0,Y 332.757,Z 984.44,A -85,B 0,C 180,E1 -14482.112,E2 -14482.112} C_VEL
LIN {X 0,Y 332.801,Z 988.228,A -85,B 0,C 180,E1 -14483.941,E2 -14483.941} C_VEL
LIN {X 0,Y 332.945,Z 990.199,A -85,B 0,C 180,E1 -14485.159,E2 -14485.159} C_VEL
LIN {X 0,Y 333.046,Z 991.676,A -85,B 0,C 180,E1 -14486.373,E2 -14486.373} C_VEL
LIN {X 0,Y 333.096,Z 992.725,A -85,B 0,C 180,E1 -14487.584,E2 -14487.584} C_VEL
LIN {X 0,Y 333.173,Z 993.371,A -85,B 0,C 180,E1 -14488.793,E2 -14488.793} C_VEL
LIN {X 0,Y 333.239,Z 993.604,A -85,B 0,C 180,E1 -14490.002,E2 -14490.002} C_VEL
LIN {X 0,Y 333.174,Z 993.365,A -85,B 0,C 180,E1 -14491.211,E2 -14491.211} C_VEL
LIN {X 0,Y 333.097,Z 992.714,A -85,B 0,C 180,E1 -14492.421,E2 -14492.421} C_VEL
LIN {X 0,Y 333.047,Z 991.66,A -85,B 0,C 180,E1 -14493.632,E2 -14493.632} C_VEL
LIN {X 0,Y 332.945,Z 990.176,A -85,B 0,C 180,E1 -14494.846,E2 -14494.846} C_VEL
LIN {X 0,Y 332.796,Z 986.399,A -85,B 0,C 180,E1 -14496.998,E2 -14496.998} C_VEL
LIN {X 0,Y 332.799,Z 981.245,A -85,B 0,C 180,E1 -14499.115,E2 -14499.115} C_VEL
LIN {X 0,Y 333.07,Z 975.497,A -85,B 0,C 180,E1 -14500.949,E2 -14500.949} C_VEL
LIN {X 0,Y 333.703,Z 968.384,A -85,B 0,C 180,E1 -14502.778,E2 -14502.778} C_VEL
LIN {X 0,Y 334.647,Z 959.525,A -85,B 0,C 180,E1 -14504.599,E2 -14504.599} C_VEL
LIN {X 0,Y 335.798,Z 949.512,A -85,B 0,C 180,E1 -14506.258,E2 -14506.258} C_VEL
LIN {X 0,Y 337.731,Z 936.07,A -85,B 0,C 180,E1 -14508.19,E2 -14508.19} C_VEL
LIN {X 0,Y 337.931,Z 925.203,A -85,B 0,C 180,E1 -14509.556,E2 -14509.556} C_VEL
LIN {X 0,Y 338.251,Z 913.743,A -85,B 0,C 180,E1 -14510.774,E2 -14510.774} C_VEL
LIN {X 0,Y 338.339,Z 904.483,A -85,B 0,C 180,E1 -14511.637,E2 -14511.637} C_VEL
LIN {X 0,Y 337.17,Z 892.385,A -85,B 0,C 180,E1 -14512.718,E2 -14512.718} C_VEL
LIN {X 0,Y 334.995,Z 879.466,A -85,B 0,C 180,E1 -14513.812,E2 -14513.812} C_VEL
LIN {X 0,Y 334.158,Z 875.352,A -85,B 0,C 180,E1 -14514.153,E2 -14514.153} C_VEL
LIN {X 0,Y 334.145,Z 874.641,A -85,B 0,C 180,E1 -14514.216,E2 -14514.216} C_VEL
LIN {X 0,Y 335.2,Z 862.81,A -85,B 0,C 180,E1 -14518.285,E2 -14518.285} C_VEL
LIN {X 0,Y 336.361,Z 851.48,A -85,B 0,C 180,E1 -14522.197,E2 -14522.197} C_VEL
LIN {X 0,Y 337.602,Z 841.415,A -85,B 0,C 180,E1 -14525.72,E2 -14525.72} C_VEL
LIN {X 0,Y 338.297,Z 835.417,A -85,B 0,C 180,E1 -14527.867,E2 -14527.867} C_VEL
LIN {X 0,Y 337.311,Z 829.335,A -85,B 0,C 180,E1 -14530.235,E2 -14530.235} C_VEL
LIN {X 0,Y 336.051,Z 822.685,A -85,B 0,C 180,E1 -14532.948,E2 -14532.948} C_VEL
LIN {X 0,Y 334.219,Z 813.693,A -85,B 0,C 180,E1 -14536.879,E2 -14536.879} C_VEL
LIN {X 0,Y 333.621,Z 810.928,A -85,B 0,C 180,E1 -14538.225,E2 -14538.225} C_VEL
LIN {X 0,Y 333.647,Z 810.926,A -85,B 0,C 180,E1 -14542.348,E2 -14542.348} C_VEL
LIN {X 0,Y 333.678,Z 810.919,A -85,B 0,C 180,E1 -14545.342,E2 -14545.342} C_VEL
LIN {X 0,Y 333.633,Z 810.926,A -85,B 0,C 180,E1 -14548.222,E2 -14548.222} C_VEL
LIN {X 0,Y 333.63,Z 810.929,A -85,B 0,C 180,E1 -14551.02,E2 -14551.02} C_VEL
LIN {X 0,Y 333.661,Z 810.924,A -85,B 0,C 180,E1 -14554.924,E2 -14554.924} C_VEL
LIN {X 0,Y 333.691,Z 810.965,A -85,B 0,C 180,E1 -14555.607,E2 -14555.607} C_VEL
LIN {X 0,Y 334.682,Z 813.776,A -85,B 0,C 180,E1 -14555.976,E2 -14555.976} C_VEL
LIN {X 0,Y 339.146,Z 821.882,A -85,B 0,C 180,E1 -14557.361,E2 -14557.361} C_VEL
LIN {X 0,Y 343.463,Z 832.215,A -85,B 0,C 180,E1 -14559.016,E2 -14559.016} C_VEL
LIN {X 0,Y 345.622,Z 839.648,A -85,B 0,C 180,E1 -14560.192,E2 -14560.192} C_VEL
LIN {X 0,Y 345.733,Z 841.917,A -85,B 0,C 180,E1 -14560.52,E2 -14560.52} C_VEL
LIN {X 0,Y 344.428,Z 851.188,A -85,B 0,C 180,E1 -14561.716,E2 -14561.716} C_VEL
LIN {X 0,Y 343.308,Z 857.966,A -85,B 0,C 180,E1 -14562.732,E2 -14562.732} C_VEL
LIN {X 0,Y 341.87,Z 866.177,A -85,B 0,C 180,E1 -14564.194,E2 -14564.194} C_VEL
LIN {X 0,Y 340.482,Z 872.885,A -85,B 0,C 180,E1 -14565.659,E2 -14565.659} C_VEL
LIN {X 0,Y 339.323,Z 878.659,A -85,B 0,C 180,E1 -14567.176,E2 -14567.176} C_VEL
LIN {X 0,Y 338.282,Z 883.23,A -85,B 0,C 180,E1 -14568.617,E2 -14568.617} C_VEL
LIN {X 0,Y 337.104,Z 887.829,A -85,B 0,C 180,E1 -14570.399,E2 -14570.399} C_VEL
LIN {X 0,Y 336.449,Z 890.222,A -85,B 0,C 180,E1 -14571.592,E2 -14571.592} C_VEL
LIN {X 0,Y 335.761,Z 892.112,A -85,B 0,C 180,E1 -14572.785,E2 -14572.785} C_VEL
LIN {X 0,Y 335.052,Z 894.667,A -85,B 0,C 180,E1 -14575.187,E2 -14575.187} C_VEL
LIN {X 0,Y 334.462,Z 895.536,A -85,B 0,C 180,E1 -14577.591,E2 -14577.591} C_VEL
LIN {X 0,Y 334.187,Z 895.383,A -85,B 0,C 180,E1 -14578.795,E2 -14578.795} C_VEL
LIN {X 0,Y 333.934,Z 894.785,A -85,B 0,C 180,E1 -14580,E2 -14580} C_VEL
LIN {X 0,Y 333.807,Z 892.375,A -85,B 0,C 180,E1 -14582.413,E2 -14582.413} C_VEL
LIN {X 0,Y 333.776,Z 889.434,A -85,B 0,C 180,E1 -14584.226,E2 -14584.226} C_VEL
LIN {X 0,Y 334.183,Z 885.424,A -85,B 0,C 180,E1 -14586.036,E2 -14586.036} C_VEL
LIN {X 0,Y 334.605,Z 879.251,A -85,B 0,C 180,E1 -14588.151,E2 -14588.151} C_VEL
LIN {X 0,Y 335.023,Z 872.609,A -85,B 0,C 180,E1 -14589.966,E2 -14589.966} C_VEL
LIN {X 0,Y 335.557,Z 866.026,A -85,B 0,C 180,E1 -14591.477,E2 -14591.477} C_VEL
LIN {X 0,Y 336.134,Z 857.926,A -85,B 0,C 180,E1 -14592.989,E2 -14592.989} C_VEL
LIN {X 0,Y 336.705,Z 850.392,A -85,B 0,C 180,E1 -14594.197,E2 -14594.197} C_VEL
LIN {X 0,Y 337.262,Z 842.762,A -85,B 0,C 180,E1 -14595.253,E2 -14595.253} C_VEL
LIN {X 0,Y 337.994,Z 832.946,A -85,B 0,C 180,E1 -14596.417,E2 -14596.417} C_VEL
LIN {X 0,Y 338.113,Z 828.1,A -85,B 0,C 180,E1 -14596.918,E2 -14596.918} C_VEL
LIN {X 0,Y 335.129,Z 816.433,A -85,B 0,C 180,E1 -14598.077,E2 -14598.077} C_VEL
LIN {X 0,Y 333.712,Z 810.913,A -85,B 0,C 180,E1 -14598.554,E2 -14598.554} C_VEL
LIN {X 0,Y 333.648,Z 810.919,A -85,B 0,C 180,E1 -14602.281,E2 -14602.281} C_VEL
LIN {X 0,Y 333.662,Z 810.92,A -85,B 0,C 180,E1 -14605.077,E2 -14605.077} C_VEL
LIN {X 0,Y 333.636,Z 810.919,A -85,B 0,C 180,E1 -14608.979,E2 -14608.979} C_VEL
LIN {X 0,Y 333.651,Z 810.911,A -85,B 0,C 180,E1 -14612.586,E2 -14612.586} C_VEL
LIN {X 0,Y 333.68,Z 810.916,A -85,B 0,C 180,E1 -14616.139,E2 -14616.139} C_VEL
LIN {X 0,Y 333.608,Z 810.924,A -85,B 0,C 180,E1 -14619.198,E2 -14619.198} C_VEL
LIN {X 0,Y 333.636,Z 810.921,A -85,B 0,C 180,E1 -14622.498,E2 -14622.498} C_VEL
LIN {X 0,Y 333.603,Z 810.927,A -85,B 0,C 180,E1 -14625.954,E2 -14625.954} C_VEL
LIN {X 0,Y 333.609,Z 810.927,A -85,B 0,C 180,E1 -14629.323,E2 -14629.323} C_VEL
LIN {X 0,Y 333.669,Z 810.916,A -85,B 0,C 180,E1 -14633.167,E2 -14633.167} C_VEL
LIN {X 0,Y 333.681,Z 810.918,A -85,B 0,C 180,E1 -14635.34,E2 -14635.34} C_VEL
LIN {X 0,Y 333.697,Z 810.913,A -85,B 0,C 180,E1 -14639.636,E2 -14639.636} C_VEL
LIN {X 0,Y 333.746,Z 810.907,A -85,B 0,C 180,E1 -14642.399,E2 -14642.399} C_VEL
LIN {X 0,Y 333.733,Z 810.903,A -85,B 0,C 180,E1 -14645.089,E2 -14645.089} C_VEL
LIN {X 0,Y 333.717,Z 811.013,A -85,B 0,C 180,E1 -14649.038,E2 -14649.038} C_VEL
LIN {X 0,Y 337.782,Z 822.468,A -85,B 0,C 180,E1 -14650.14,E2 -14650.14} C_VEL
LIN {X 0,Y 341.133,Z 833.425,A -85,B 0,C 180,E1 -14651.387,E2 -14651.387} C_VEL
LIN {X 0,Y 341.625,Z 835.301,A -85,B 0,C 180,E1 -14651.616,E2 -14651.616} C_VEL
LIN {X 0,Y 340.548,Z 846.471,A -85,B 0,C 180,E1 -14652.896,E2 -14652.896} C_VEL
LIN {X 0,Y 339.42,Z 856.81,A -85,B 0,C 180,E1 -14654.383,E2 -14654.383} C_VEL
LIN {X 0,Y 338.382,Z 865.173,A -85,B 0,C 180,E1 -14655.873,E2 -14655.873} C_VEL
LIN {X 0,Y 337.206,Z 873.291,A -85,B 0,C 180,E1 -14657.663,E2 -14657.663} C_VEL
LIN {X 0,Y 336.313,Z 879.852,A -85,B 0,C 180,E1 -14659.477,E2 -14659.477} C_VEL
LIN {X 0,Y 335.5,Z 885.762,A -85,B 0,C 180,E1 -14661.566,E2 -14661.566} C_VEL
LIN {X 0,Y 334.719,Z 889.655,A -85,B 0,C 180,E1 -14663.367,E2 -14663.367} C_VEL
LIN {X 0,Y 334.274,Z 892.507,A -85,B 0,C 180,E1 -14665.174,E2 -14665.174} C_VEL
LIN {X 0,Y 334.273,Z 893.845,A -85,B 0,C 180,E1 -14666.382,E2 -14666.382} C_VEL
LIN {X 0,Y 333.995,Z 895.422,A -85,B 0,C 180,E1 -14668.792,E2 -14668.792} C_VEL
LIN {X 0,Y 333.95,Z 895.653,A -85,B 0,C 180,E1 -14669.998,E2 -14669.998} C_VEL
LIN {X 0,Y 334.119,Z 894.889,A -85,B 0,C 180,E1 -14672.409,E2 -14672.409} C_VEL
LIN {X 0,Y 334.225,Z 893.953,A -85,B 0,C 180,E1 -14673.615,E2 -14673.615} C_VEL
LIN {X 0,Y 334.262,Z 892.655,A -85,B 0,C 180,E1 -14674.822,E2 -14674.822} C_VEL
LIN {X 0,Y 334.707,Z 889.849,A -85,B 0,C 180,E1 -14676.629,E2 -14676.629} C_VEL
LIN {X 0,Y 335.521,Z 886.009,A -85,B 0,C 180,E1 -14678.429,E2 -14678.429} C_VEL
LIN {X 0,Y 336.206,Z 881.579,A -85,B 0,C 180,E1 -14680.065,E2 -14680.065} C_VEL
LIN {X 0,Y 336.968,Z 874.933,A -85,B 0,C 180,E1 -14682.036,E2 -14682.036} C_VEL
LIN {X 0,Y 338.111,Z 867.157,A -85,B 0,C 180,E1 -14683.827,E2 -14683.827} C_VEL
LIN {X 0,Y 339.136,Z 859.229,A -85,B 0,C 180,E1 -14685.318,E2 -14685.318} C_VEL
LIN {X 0,Y 340.26,Z 849.537,A -85,B 0,C 180,E1 -14686.806,E2 -14686.806} C_VEL
LIN {X 0,Y 341.224,Z 839.983,A -85,B 0,C 180,E1 -14687.993,E2 -14687.993} C_VEL
LIN {X 0,Y 341.71,Z 836.086,A -85,B 0,C 180,E1 -14688.398,E2 -14688.398} C_VEL
LIN {X 0,Y 339.259,Z 827.064,A -85,B 0,C 180,E1 -14689.47,E2 -14689.47} C_VEL
LIN {X 0,Y 335.769,Z 816.731,A -85,B 0,C 180,E1 -14690.548,E2 -14690.548} C_VEL
LIN {X 0,Y 333.745,Z 810.91,A -85,B 0,C 180,E1 -14691.087,E2 -14691.087} C_VEL
LIN {X 0,Y 333.715,Z 810.915,A -85,B 0,C 180,E1 -14695.099,E2 -14695.099} C_VEL
